CASE eHomeSeq OF
    E_HomingRoutines.eHomeToRef_Bwd:
        stDetectDirection := mcNegativeDirection;
        fbFinishHoming.Distance := fHomeFinishDistance;
    E_HomingRoutines.eHomeToRef_Fwd:
        stDetectDirection := mcPositiveDirection;
        fbFinishHoming.Distance := -fHomeFinishDistance;
END_CASE
bViaLimitSwitch := FALSE;

fbStepAbsoluteSwitchDetection.Options.DisableDriveAccess := stOptions.DisableDriveAccess;
fbStepAbsoluteSwitchDetection(
    Axis := Axis,
    Execute := bDetectionFB_Execute,
    Parameter := stHomingParameter,
    Direction := stDetectDirection,
    SwitchMode := stConfig.stHomingConfig.eRefSwitchMode,
    ReferenceSignal := stRefSwitchSignal,
    Velocity := fVelocityFromCam,
    PositiveLimitSwitch := NOT(bLimitFwd),
    NegativeLimitSwitch := NOT(bLimitBwd),
    Options := stOptions,
    Done => bDetectionFB_Done,
    Busy => bDetectionFB_Busy,
    CommandAborted => bDetectionFB_CommandAborted,
    Error => bDetectionFB_Error,
    ErrorID => nDetectionFB_ErrorID,
    RecordedPosition => fRecordedPosition);
END_ACTION

END_FUNCTION_BLOCK

// ---- tc_mca_std_lib/POUs/Pneumatics/FB_PneumaticAxis.TcPOU

FUNCTION_BLOCK FB_PneumaticAxis

VAR_IN_OUT
    stPneumaticAxisStruct: ST_PneumaticAxisStruct;
END_VAR
VAR
    fbTimerExtend: TON; //Timing the extraction of the cylinder
    fbTimerRetract: TON; //Timing the retraction of the cylinder
    fbTrigRisingEdgePermit: R_TRIG; //Rising edge detection for Permit signal
    fbTrigExtendManual: R_TRIG; //Rising edge detection for manual push button
    fbTrigRetractManual: R_TRIG; //Rising edge detection for manual push button
    bStateChange: BOOL := FALSE; //State of the cylinder changed from extend to retract and vice versa
    bStartExtendManual: BOOL; //Variable to control the solenoid valve with momentary push button
    bStartRetractManual: BOOL; //VAriable to control the solenoid valve with momentary push button
END_VAR


Initialization();

CASE stPneumaticAxisStruct.ePneumaticAxisMode OF

    E_PneumaticMode.eSingleSolenoidControl:
    Single_Solenoid();

    E_PneumaticMode.eError:
    Single_Solenoid_Error();

    E_PneumaticMode.eReset:
    Reset();
END_CASE

ACTION ErrorCheck:
//IF the command to extract is given, but the cylinder hasn't moved from the bEndSwitchBwd
    IF  fbTimerExtend.Q AND stPneumaticAxisStruct.stPneumaticAxisStatus.bRetracted THEN
             stPneumaticAxisStruct.stPneumaticAxisStatus.bExtending := FALSE;
             stPneumaticAxisStruct.ePneumaticAxisMode := E_PneumaticMode.eError;
    END_IF
//If the command to extract has timed out
    IF  fbTimerExtend.Q AND (NOT stPneumaticAxisStruct.stPneumaticAxisStatus.bRetracted AND NOT stPneumaticAxisStruct.stPneumaticAxisStatus.bExtended) THEN
            stPneumaticAxisStruct.stPneumaticAxisStatus.bExtending := FALSE;
            stPneumaticAxisStruct.ePneumaticAxisMode := E_PneumaticMode.eError;
    END_IF

//IF the command to retract has been given, but the cylinder hasn't moved from bEndSwitchFwd
        IF  fbTimerRetract.Q AND stPneumaticAxisStruct.stPneumaticAxisStatus.bExtended THEN
            stPneumaticAxisStruct.stPneumaticAxisStatus.bRetracting := FALSE;
            stPneumaticAxisStruct.ePneumaticAxisMode := E_PneumaticMode.eError;
        END_IF

//If the command to retract has timed out
        IF  fbTimerRetract.Q AND (NOT stPneumaticAxisStruct.stPneumaticAxisStatus.bExtended AND NOT stPneumaticAxisStruct.stPneumaticAxisStatus.bRetracted) THEN
            stPneumaticAxisStruct.stPneumaticAxisStatus.bRetracting := FALSE;
            stPneumaticAxisStruct.ePneumaticAxisMode := E_PneumaticMode.eError;
        END_IF
END_ACTION

ACTION Initialization:
//Set the inputs of limit switches to bExtracted and bRetracted states of the pneumatic cylinders
stPneumaticAxisStruct.stPneumaticAxisStatus.bRetracted := stPneumaticAxisStruct.stPneumaticAxisInputs.bEndSwitchBwd;
stPneumaticAxisStruct.stPneumaticAxisStatus.bExtended := stPneumaticAxisStruct.stPneumaticAxisInputs.bEndSwitchFwd;
stPneumaticAxisStruct.stPneumaticAxisStatus.bSolenoidActive := stPneumaticAxisStruct.stPneumaticAxisInputs.bSolenoidActive;
stPneumaticAxisStruct.stPneumaticAxisStatus.bPSSPermitOK := stPneumaticAxisStruct.stPneumaticAxisInputs.bPSSPermit;
stPneumaticAxisStruct.stPneumaticAxisStatus.bInterlocked := stPneumaticAxisStruct.stPneumaticAxisControl.bInterlock;


//Check if Permit signal is ON
IF NOT stPneumaticAxisStruct.stPneumaticAxisInputs.bPSSPermit THEN
            stPneumaticAxisStruct.stPneumaticAxisOutputs.bValveOn := FALSE;
            stPneumaticAxisStruct.ePneumaticAxisMode := E_PneumaticMode.eError;
END_IF

//Reset Error
fbTrigRisingEdgePermit(clk:=stPneumaticAxisStruct.stPneumaticAxisControl.bReset);

IF fbTrigRisingEdgePermit.Q THEN
    stPneumaticAxisStruct.ePneumaticAxisMode := E_PneumaticMode.eReset;
END_IF

//Check if Interlock signal is ON
IF stPneumaticAxisStruct.stPneumaticAxisControl.bInterlock THEN
            stPneumaticAxisStruct.stPneumaticAxisOutputs.bValveOn := FALSE;
            stPneumaticAxisStruct.ePneumaticAxisMode := E_PneumaticMode.eError;
END_IF

//Check for errors in Air pressure (to be implemented)
END_ACTION

ACTION Reset:
//Reset all the error messages
//Set the operating mode to Single Solenoid Control

stPneumaticAxisStruct.stPneumaticAxisStatus.sStatus := 'NO_ERRORS_READY_TO_START';
stPneumaticAxisStruct.ePneumaticAxisErrors := E_PneumaticAxisErrors.eNoError;
stPneumaticAxisStruct.stPneumaticAxisStatus.bError := FALSE;
stPneumaticAxisStruct.ePneumaticAxisMode := E_PneumaticMode.eSingleSolenoidControl;
END_ACTION

ACTION Single_Solenoid:
//Enter allowed times for extraction and retraction of pneumatic cylinder in seconds
 fbTimerExtend.PT := INT_TO_TIME( stPneumaticAxisStruct.stPneumaticAxisConfig.nTimeToExtend)*1000;
 fbTimerRetract.PT := INT_TO_TIME( stPneumaticAxisStruct.stPneumaticAxisConfig.nTimeToRetract)*1000;


//Starting the timing of extraction movement
fbTimerExtend();
fbTimerExtend(IN := stPneumaticAxisStruct.stPneumaticAxisStatus.bExtending);

//If the manual momentary push button is used for control of the pneumatic cylinder
fbTrigExtendManual(clk:=stPneumaticAxisStruct.stPneumaticAxisInputs.bOpenManual);

IF fbTrigExtendManual.Q THEN
    bStartExtendManual := TRUE;
END_IF

//Starting the extraction movement
IF (stPneumaticAxisStruct.stPneumaticAxisControl.bExtend OR bStartExtendManual) THEN
        stPneumaticAxisStruct.stPneumaticAxisOutputs.bValveOn := TRUE;
        stPneumaticAxisStruct.stPneumaticAxisStatus.bExtending := TRUE;
//If the command to retract is given while the cylinder is extracting
    IF NOT stPneumaticAxisStruct.stPneumaticAxisStatus.bExtended AND NOT stPneumaticAxisStruct.stPneumaticAxisStatus.bRetracted THEN
        IF (stPneumaticAxisStruct.stPneumaticAxisControl.bRetract OR bStartRetractManual) THEN
            stPneumaticAxisStruct.stPneumaticAxisOutputs.bValveOn := FALSE;
            stPneumaticAxisStruct.stPneumaticAxisStatus.bRetracting := TRUE;
            stPneumaticAxisStruct.stPneumaticAxisStatus.bExtending := FALSE;
            stPneumaticAxisStruct.stPneumaticAxisControl.bExtend := FALSE;
        bStartExtendManual := FALSE;
        END_IF
    END_IF


END_IF
//Check for errors while the cylinder is extending
ErrorCheck();

// Extraction of the cylinder finished, reset timer
IF (stPneumaticAxisStruct.stPneumaticAxisControl.bExtend OR bStartExtendManual) AND stPneumaticAxisStruct.stPneumaticAxisStatus.bExtended THEN
        bStateChange := TRUE;
        stPneumaticAxisStruct.stPneumaticAxisStatus.bExtending := FALSE;
        stPneumaticAxisStruct.stPneumaticAxisControl.bExtend := FALSE;
        bStartExtendManual := FALSE;
END_IF



//Starting the retraction movement and retraction timing
fbTimerRetract();
fbTimerRetract (IN := stPneumaticAxisStruct.stPneumaticAxisStatus.bRetracting);

//If the manual momentary push button is used for control of the pneumatic cylinder
fbTrigRetractManual(clk:=stPneumaticAxisStruct.stPneumaticAxisInputs.bCloseManual);

IF fbTrigRetractManual.Q THEN
    bStartRetractManual := TRUE;
END_IF

IF (stPneumaticAxisStruct.stPneumaticAxisControl.bRetract OR bStartRetractManual) THEN
        stPneumaticAxisStruct.stPneumaticAxisOutputs.bValveOn := FALSE;
        stPneumaticAxisStruct.stPneumaticAxisStatus.bRetracting := TRUE;


END_IF
//Check for errors while the cylinder is retracting
ErrorCheck();
// Retraction of the cylinder finished, reset timer
IF  (stPneumaticAxisStruct.stPneumaticAxisControl.bRetract OR bStartRetractManual) AND stPneumaticAxisStruct.stPneumaticAxisStatus.bRetracted THEN
        bStateChange := FALSE;
        stPneumaticAxisStruct.stPneumaticAxisStatus.bRetracting := FALSE;
        stPneumaticAxisStruct.stPneumaticAxisControl.bRetract := FALSE;
        bStartRetractManual := FALSE;
END_IF
END_ACTION

ACTION Single_Solenoid_Error:
IF NOT stPneumaticAxisStruct.stPneumaticAxisInputs.bPSSPermit THEN
    stPneumaticAxisStruct.ePneumaticAxisErrors := E_PneumaticAxisErrors.eNoPSSPermit;
END_IF

IF stPneumaticAxisStruct.stPneumaticAxisControl.bInterlock THEN
     stPneumaticAxisStruct.ePneumaticAxisErrors := E_PneumaticAxisErrors.eInterlockOn;
END_IF

IF  fbTimerExtend.Q AND stPneumaticAxisStruct.stPneumaticAxisStatus.bRetracted THEN
    stPneumaticAxisStruct.ePneumaticAxisErrors := E_PneumaticAxisErrors.eNotMovingExtract;
END_IF

IF  fbTimerExtend.Q AND NOT stPneumaticAxisStruct.stPneumaticAxisStatus.bRetracted AND NOT stPneumaticAxisStruct.stPneumaticAxisStatus.bExtended THEN
    stPneumaticAxisStruct.ePneumaticAxisErrors := E_PneumaticAxisErrors.eExtractTimedOut;
END_IF

IF  fbTimerRetract.Q AND stPneumaticAxisStruct.stPneumaticAxisStatus.bExtended THEN
    stPneumaticAxisStruct.ePneumaticAxisErrors := E_PneumaticAxisErrors.eNotMovingRetract;
END_IF

IF  fbTimerRetract.Q AND NOT stPneumaticAxisStruct.stPneumaticAxisStatus.bExtended AND NOT stPneumaticAxisStruct.stPneumaticAxisStatus.bRetracted THEN
    stPneumaticAxisStruct.ePneumaticAxisErrors := E_PneumaticAxisErrors.eRetractTimedOut;
END_IF


CASE  stPneumaticAxisStruct.ePneumaticAxisErrors OF

    E_PneumaticAxisErrors.eNoError:
    stPneumaticAxisStruct.stPneumaticAxisStatus.bError := FALSE;

    E_PneumaticAxisErrors.eExtractTimedOut:
    stPneumaticAxisStruct.stPneumaticAxisStatus.sStatus := 'ERROR: COMMAND TIMED OUT';
    stPneumaticAxisStruct.stPneumaticAxisStatus.bError := TRUE;

    E_PneumaticAxisErrors.eRetractTimedOut:
    stPneumaticAxisStruct.stPneumaticAxisStatus.sStatus := 'ERROR: COMMAND TIMED OUT';
    stPneumaticAxisStruct.stPneumaticAxisStatus.bError := TRUE;

    E_PneumaticAxisErrors.eNotMovingExtract:
    stPneumaticAxisStruct.stPneumaticAxisStatus.sStatus := 'ERROR: CYLINDER NOT MOVING';
    stPneumaticAxisStruct.stPneumaticAxisStatus.bError := TRUE;

    E_PneumaticAxisErrors.eNotMovingRetract:
    stPneumaticAxisStruct.stPneumaticAxisStatus.sStatus := 'ERROR: CYLINDER NOT MOVING';
    stPneumaticAxisStruct.stPneumaticAxisStatus.bError := TRUE;

    E_PneumaticAxisErrors.eNoPSSPermit:
    stPneumaticAxisStruct.stPneumaticAxisStatus.sStatus := 'ERROR: NO PERMIT SIGNAL';
    stPneumaticAxisStruct.stPneumaticAxisStatus.bError := TRUE;

    E_PneumaticAxisErrors.eInterlockOn:
    stPneumaticAxisStruct.stPneumaticAxisStatus.sStatus := 'ERROR: INTERLOCK SIGNAL ON';
    stPneumaticAxisStruct.stPneumaticAxisStatus.bError := TRUE;

END_CASE

stPneumaticAxisStruct.stPneumaticAxisControl.bExtend := FALSE;
stPneumaticAxisStruct.stPneumaticAxisControl.bRetract := FALSE;
stPneumaticAxisStruct.stPneumaticAxisOutputs.bValveOn := FALSE;
bStartExtendManual := FALSE;
bStartRetractManual := FALSE;
stPneumaticAxisStruct.stPneumaticAxisStatus.bExtending := FALSE;
stPneumaticAxisStruct.stPneumaticAxisStatus.bRetracting := FALSE;
END_ACTION

END_FUNCTION_BLOCK

// ---- POUs/Application_Specific/Axes/Axis_Template.TcPOU
PROGRAM Axis_Template
VAR
//Outputs: Power for Limit switches, Home Sensors, etc.
    //bPowerSwitchesAxis1 AT %Q*: BOOL:= TRUE;

//Hardware interlocks
    //bInterlockFwdOK AT %I*: BOOL;
END_VAR

//Initial parameters of an Axis
(* Uncomment the next IF statement to configure and activate the intial parameters of the axis
IF _TaskInfo[fbGetCurTaskIndex.index].FirstCycle THEN
    //Axis description for EPICS PV
    GVL.astAxes[x].stDescription.sAxisName := 'MotorApplication1';
    GVL.astAxes[x].stDescription.eUnit := E_AxisEngUnit.eMeter;
    GVL.astAxes[x].stDescription.nPrefix := -3;

    //Initial default values:
    GVL.astAxes[x].stConfig.eHomeSeq := 0;
    GVL.astAxes[x].stConfig.fHomePosition := 0.0;
    GVL.astAxes[x].stConfig.fHomeFinishDistance := 0.0;
    GVL.astAxes[x].stConfig.eRestorePosition := E_RestorePosition.eRestoreWithoutHome;

    GVL.astAxes[x].stConfig.bEnableTemperatureDisable := FALSE;
    GVL.astAxes[x].stConfig.fMaxTemperature := 0.0;
END_IF
*)
//Define ACTIONS() or write exclusive code for an specific axis.
(*Eg. Stop when temperature reaches certain values, reduce speed if  a signal is activated, etc.
Eg. GVL.astAxes[x].stControl.bInterlockFwd := NOT bInterlockFwdOK;*)

END_PROGRAM

// ---- POUs/Application_Specific/Applications/Application_Template.TcPOU
PROGRAM Application_Template
VAR
    //Define all necessary variables for your application

END_VAR

//Program any specific code or safety code for an specific application when it involves multiple axes
//Eg. Collision avoidance, interlocks, sequencing, etc.

END_PROGRAM

// ---- POUs/Application_Specific/Axes/Pneumatics_Template.TcPOU
PROGRAM Pneumatics_Template
VAR
END_VAR

//Test the program to control pneumatic acutator through PneumaticsVisu.
//Currently implemented control of single solenoid through PLC and and manually, with two momentary push buttons.

END_PROGRAM

// ---- tc_mca_std_lib/POUs/FB_ESSMonitoring.TcPOU

FUNCTION_BLOCK FB_ESSMonitoring
VAR_INPUT
    nEcMasterNetId: T_AmsNetId;
END_VAR
VAR_OUTPUT
    aErrorID: ARRAY [1..nMaxAlarms] OF INT;
    aErrorMsg: ARRAY [1..nMaxAlarms] OF STRING;
    nEcMasterFramesLost: UDINT;
    nCPULoad: UDINT;
    fCycleExecTime_ms: REAL;
    nAlarmGrpBitNumber: UDINT;
END_VAR
VAR
    //Outputs
    bFan1 AT %Q*: BOOL := TRUE;
    bFan2 AT %Q*: BOOL := TRUE;
    bDCSupplyLED AT %Q*: BOOL := TRUE;
    bAcknowledgeLED AT %Q*: BOOL;
    bStatusLED AT %Q*: BOOL;
    bWarningLED AT %Q*: BOOL;
    bEmergencyLED AT %Q*: BOOL;
    //Inputs
    b24VDC1_OK AT %I*: BOOL;
    b24VDC2_OK AT %I*: BOOL;
    b48VDC1_OK AT %I*: BOOL;
    bFuse1_OK AT %I*: BOOL;
    bFuse2_OK AT %I*: BOOL;
    bFuse3_OK AT %I*: BOOL;
    bFuse4_OK AT %I*: BOOL;
    bFuse5_OK AT %I*: BOOL;
    bFuse6_OK AT %I*: BOOL;
    bFuse7_OK AT %I*: BOOL;
    bFuse8_OK AT %I*: BOOL;
    bSafety_OK AT %I*: BOOL;
    bFan1_OK AT %I*: BOOL;
    bFan2_OK AT %I*: BOOL;
    nTemp1 AT %I*: INT;
    nTemp2 AT %I*: INT;
    nEcMasterDevState AT %I*: UINT;
    aAlarmList: ARRAY [1..nMaxAlarms] OF ST_MonitoringAlarm := [
                    (*[1]*)(nStatusLED:=E_MonitoringLedFunction.eFast, nWarningLED:=E_MonitoringLedFunction.eUndefined, nEmergencyLED:=E_MonitoringLedFunction.eSteady, nAcknowledgeLED:=E_MonitoringLedFunction.eUndefined, nErrorID:=1 ,sErrorMsg:='The DC OK Status from PS or DC-DC converter 24V-1 is OFF.'),
                    (*[2]*)(nStatusLED:=E_MonitoringLedFunction.eUndefined, nWarningLED:=E_MonitoringLedFunction.eUndefined, nEmergencyLED:=E_MonitoringLedFunction.eUndefined, nAcknowledgeLED:=E_MonitoringLedFunction.eUndefined, nErrorID:=2 ,sErrorMsg:='The DC OK Status from PS 24V-2 is OFF.'),
                    (*[3]*)(nStatusLED:=E_MonitoringLedFunction.eFast, nWarningLED:=E_MonitoringLedFunction.eUndefined, nEmergencyLED:=E_MonitoringLedFunction.eSteady, nAcknowledgeLED:=E_MonitoringLedFunction.eUndefined, nErrorID:=4 ,sErrorMsg:='The DC OK Status from PS 48V-1 is OFF.'),
                    (*[4]*)(nStatusLED:=E_MonitoringLedFunction.eUndefined, nWarningLED:=E_MonitoringLedFunction.eUndefined, nEmergencyLED:=E_MonitoringLedFunction.eUndefined, nAcknowledgeLED:=E_MonitoringLedFunction.eUndefined, nErrorID:=8 ,sErrorMsg:='Output 1 on LOCC box 1 tripped'),
                    (*[5]*)(nStatusLED:=E_MonitoringLedFunction.eSlow, nWarningLED:=E_MonitoringLedFunction.eUndefined, nEmergencyLED:=E_MonitoringLedFunction.eSteady, nAcknowledgeLED:=E_MonitoringLedFunction.eUndefined, nErrorID:=9 ,sErrorMsg:='Output 2 on LOCC box 1 tripped'),
                    (*[6]*)(nStatusLED:=E_MonitoringLedFunction.eUndefined, nWarningLED:=E_MonitoringLedFunction.eUndefined, nEmergencyLED:=E_MonitoringLedFunction.eUndefined, nAcknowledgeLED:=E_MonitoringLedFunction.eUndefined, nErrorID:=10 ,sErrorMsg:='Output 1 on LOCC box 2 tripped'),
                    (*[7]*)(nStatusLED:=E_MonitoringLedFunction.eSlow, nWarningLED:=E_MonitoringLedFunction.eUndefined, nEmergencyLED:=E_MonitoringLedFunction.eSteady, nAcknowledgeLED:=E_MonitoringLedFunction.eUndefined, nErrorID:=11 ,sErrorMsg:='Output 2 on LOCC box 2 tripped'),
                    (*[8]*)(nStatusLED:=E_MonitoringLedFunction.eSteady, nWarningLED:=E_MonitoringLedFunction.eSteady, nEmergencyLED:=E_MonitoringLedFunction.eUndefined, nAcknowledgeLED:=E_MonitoringLedFunction.eUndefined, nErrorID:=12 ,sErrorMsg:='Output 1 on LOCC box 3 tripped'),
                    (*[9]*)(nStatusLED:=E_MonitoringLedFunction.eSteady, nWarningLED:=E_MonitoringLedFunction.eSteady, nEmergencyLED:=E_MonitoringLedFunction.eUndefined, nAcknowledgeLED:=E_MonitoringLedFunction.eUndefined, nErrorID:=13 ,sErrorMsg:='Output 2 on LOCC box 3 tripped'),
                    (*[10]*)(nStatusLED:=E_MonitoringLedFunction.eSlow, nWarningLED:=E_MonitoringLedFunction.eSteady, nEmergencyLED:=E_MonitoringLedFunction.eUndefined, nAcknowledgeLED:=E_MonitoringLedFunction.eUndefined, nErrorID:=14 ,sErrorMsg:='LOCC box 4 or single DC breaker 1 tripped'),
                    (*[11]*)(nStatusLED:=E_MonitoringLedFunction.eSlow, nWarningLED:=E_MonitoringLedFunction.eSteady, nEmergencyLED:=E_MonitoringLedFunction.eUndefined, nAcknowledgeLED:=E_MonitoringLedFunction.eUndefined, nErrorID:=15 ,sErrorMsg:='LOCC box 5 or single DC breaker 2 tripped'),
                    (*[12]*)(nStatusLED:=E_MonitoringLedFunction.eUndefined, nWarningLED:=E_MonitoringLedFunction.eSteady, nEmergencyLED:=E_MonitoringLedFunction.eUndefined, nAcknowledgeLED:=E_MonitoringLedFunction.eUndefined, nErrorID:=21 ,sErrorMsg:='Speed of Fan 1 below a critical limit'),
                    (*[13]*)(nStatusLED:=E_MonitoringLedFunction.eUndefined, nWarningLED:=E_MonitoringLedFunction.eSteady, nEmergencyLED:=E_MonitoringLedFunction.eUndefined, nAcknowledgeLED:=E_MonitoringLedFunction.eUndefined, nErrorID:=22 ,sErrorMsg:='Speed of Fan 2 below a critical limit'),
                    (*[14]*)(nStatusLED:=E_MonitoringLedFunction.eUndefined, nWarningLED:=E_MonitoringLedFunction.eSteady, nEmergencyLED:=E_MonitoringLedFunction.eSteady, nAcknowledgeLED:=E_MonitoringLedFunction.eUndefined, nErrorID:=23 ,sErrorMsg:='Temperature 1 too high' ),
                    (*[15]*)(nStatusLED:=E_MonitoringLedFunction.eUndefined, nWarningLED:=E_MonitoringLedFunction.eSteady, nEmergencyLED:=E_MonitoringLedFunction.eSteady, nAcknowledgeLED:=E_MonitoringLedFunction.eUndefined, nErrorID:=24 ,sErrorMsg:='Temperature 2 too high'),
                    (*[16]*)(nStatusLED:=E_MonitoringLedFunction.eSteady, nWarningLED:=E_MonitoringLedFunction.eSteady, nEmergencyLED:=E_MonitoringLedFunction.eUndefined, nAcknowledgeLED:=E_MonitoringLedFunction.eUndefined, nErrorID:=30 ,sErrorMsg:='Safety relay 1 triggered'),
                    (*[17]*)(nStatusLED:=E_MonitoringLedFunction.eSteady, nWarningLED:=E_MonitoringLedFunction.eSlow, nEmergencyLED:=E_MonitoringLedFunction.eUndefined, nAcknowledgeLED:=E_MonitoringLedFunction.eUndefined, nErrorID:=101 ,sErrorMsg:='EtherCAT Master is not ok'),
                    (*[18]*)(nStatusLED:=E_MonitoringLedFunction.eSteady, nWarningLED:=E_MonitoringLedFunction.eSlow, nEmergencyLED:=E_MonitoringLedFunction.eSteady, nAcknowledgeLED:=E_MonitoringLedFunction.eUndefined, nErrorID:=102 ,sErrorMsg:='At least one EtherCAT slave is not in OP state'),
                    (*[19]*)(nStatusLED:=E_MonitoringLedFunction.eSteady, nWarningLED:=E_MonitoringLedFunction.eSlow, nEmergencyLED:=E_MonitoringLedFunction.eSteady, nAcknowledgeLED:=E_MonitoringLedFunction.eUndefined, nErrorID:=103 ,sErrorMsg:='At least one EtherCAT slave link is faulted'),
                    (*[20]*)(nStatusLED:=E_MonitoringLedFunction.eSteady, nWarningLED:=E_MonitoringLedFunction.eSlow, nEmergencyLED:=E_MonitoringLedFunction.eUndefined, nAcknowledgeLED:=E_MonitoringLedFunction.eUndefined, nErrorID:=104 ,sErrorMsg:='Overflow in PLC cycle time'),
                    (*[21]*)(nStatusLED:=E_MonitoringLedFunction.eSteady, nWarningLED:=E_MonitoringLedFunction.eSlow, nEmergencyLED:=E_MonitoringLedFunction.eUndefined, nAcknowledgeLED:=E_MonitoringLedFunction.eUndefined, nErrorID:=105 ,sErrorMsg:='CPU Load High')];

    aTempErrorID: ARRAY [1..nMaxAlarms] OF INT;
    aTempErrorMsg: ARRAY [1..nMaxAlarms] OF STRING;
    nLEDAlarmID: INT;
    sLEDAlarmMsg: STRING;
    nAlarmCnt: INT;
    nAlarmBitNumber: UDINT;

    bCPUOverloaded: BOOL;
    bEcMasterNotOK: BOOL;
    bSlaveStateNotOP: BOOL;
    bSlaveLinkNotOK: BOOL;
    bCycleTimeExceeded: BOOL;
    //Cpu Monitor
    fbMonitorCPU: TC_CpuUsage;
    fbUpdateCPULoadTON: TON;
    fMaxCPULoad: USINT := 85;
    //Ehtercat master device state
    bEcLinkError: BOOL;
    bEcIOlocked: BOOL;
    bEcLinkErrorRedundancyAdapter: BOOL;
    bEcMissingFrame: BOOL;
    bEcOutofSendResources: BOOL;
    bEcWatchdogTriggered: BOOL;
    bEcEthernetDriverNotFound: BOOL;
    bEcIOresetActive: BOOL;
    bEcSlaveINIT: BOOL;
    bEcSlavePreOP: BOOL;
    bEcSlaveSafeOP: BOOL;
    bEcSlaveError: BOOL;
    bEcDCnotInSync: BOOL;
    //Ehtercat slave device state
    fbUpdateEcSlaveStateTON: TON;
    fbGetEcSlaveStates: FB_EcGetAllSlaveStates;
    stSlaveState: ARRAY[0..nMaxECSlaves] OF ST_EcSlaveState;
    nActualEcSlaves: INT := 0;
    i: INT;
    //Frame statistics
    fbUpdateEcMasterFrame: TON;
    fbGetEcMasterFrames: FB_EcMasterFrameStatistic;

    nAcknowledgeLED: E_MonitoringLedFunction;
    nStatusLED: E_MonitoringLedFunction;
    nWarningLED: E_MonitoringLedFunction;
    nEmergencyLED: E_MonitoringLedFunction;
    fbFastBlinkOn: TON;
    fbFastBlinkOff: TON;
    bFastBlink: BOOL;
    fbSlowBlinkOn: TON;
    fbSlowBlinkOff: TON;
    bSlowBlink: BOOL;
END_VAR
VAR CONSTANT
    nMaxAlarms: INT := 50;
    nMaxECSlaves: INT := 255;
    nMaxTemp: INT := 10000;
END_VAR


actMonitorAlarms();
actMonitorCPU();
actMonitorEtherCAT();

ACTION actMonitorAlarms:

aAlarmList[1].bAlarmSet := NOT b24VDC1_OK;
aAlarmList[1].bAlarmReset:= TRUE;
aAlarmList[2].bAlarmSet := b24VDC2_OK;
aAlarmList[2].bAlarmReset:= TRUE;
aAlarmList[3].bAlarmSet := NOT b48VDC1_OK;
aAlarmList[3].bAlarmReset:= TRUE;
aAlarmList[4].bAlarmSet := bFuse1_OK;
aAlarmList[4].bAlarmReset:= TRUE;
aAlarmList[5].bAlarmSet :=  bFuse2_OK;
aAlarmList[5].bAlarmReset:= TRUE;
aAlarmList[6].bAlarmSet := bFuse3_OK;
aAlarmList[6].bAlarmReset:= TRUE;
aAlarmList[7].bAlarmSet := bFuse4_OK;
aAlarmList[7].bAlarmReset:= TRUE;
aAlarmList[8].bAlarmSet := bFuse5_OK;
aAlarmList[8].bAlarmReset:= TRUE;
aAlarmList[9].bAlarmSet := bFuse6_OK;
aAlarmList[9].bAlarmReset:= TRUE;
aAlarmList[10].bAlarmSet := bFuse7_OK;
aAlarmList[10].bAlarmReset:= TRUE;
aAlarmList[11].bAlarmSet := bFuse8_OK;
aAlarmList[11].bAlarmReset:= TRUE;
aAlarmList[12].bAlarmSet := NOT bFan1_OK;
aAlarmList[12].bAlarmReset:= TRUE;
aAlarmList[13].bAlarmSet := NOT bFan2_OK;
aAlarmList[13].bAlarmReset:= TRUE;
aAlarmList[14].bAlarmSet := nTemp1 > nMaxTemp;
aAlarmList[14].bAlarmReset:= TRUE;
aAlarmList[15].bAlarmSet := nTemp2 > nMaxTemp;
aAlarmList[15].bAlarmReset:= TRUE;
aAlarmList[16].bAlarmSet := NOT bSafety_OK;
aAlarmList[16].bAlarmReset:= TRUE;
aAlarmList[17].bAlarmSet := bEcMasterNotOK;
aAlarmList[17].bAlarmReset:= TRUE;
aAlarmList[18].bAlarmSet := bSlaveStateNotOP;
aAlarmList[18].bAlarmReset:= TRUE;
aAlarmList[19].bAlarmSet := bSlaveLinkNotOK;
aAlarmList[19].bAlarmReset:= TRUE;
aAlarmList[20].bAlarmSet := bCycleTimeExceeded;
aAlarmList[20].bAlarmReset:= TRUE;
aAlarmList[21].bAlarmSet := bCPUOverloaded;
aAlarmList[21].bAlarmReset:= TRUE;

FOR i:=1 TO nMaxAlarms DO
    mAlarm(stAlarmData:= aAlarmList[i]);
    IF i = 1 THEN
        nAlarmCnt := 0;
        nAlarmBitNumber := 0;
        MEMSET(ADR(aTempErrorID), 0, SIZEOF(aTempErrorID));
        MEMSET(ADR(aTempErrorMsg), 0, SIZEOF(aTempErrorMsg));
    ELSIF i = nMaxAlarms THEN
        aErrorID := aTempErrorID;
        aErrorMsg := aTempErrorMsg;
        nAlarmGrpBitNumber := nAlarmBitNumber;
    END_IF

    IF aAlarmList[i].bAlarmActive THEN
        nAlarmCnt := nAlarmCnt + 1;
        aTempErrorID[nAlarmCnt] := aAlarmList[i].nErrorID;
        aTempErrorMsg[nAlarmCnt] := aAlarmList[i].sErrorMsg;
        IF nLEDAlarmID = 0 OR (nWarningLED = E_MonitoringLedFunction.eUndefined AND nEmergencyLED = E_MonitoringLedFunction.eUndefined AND aAlarmList[i].nWarningLED > E_MonitoringLedFunction.eUndefined) OR (nEmergencyLED = E_MonitoringLedFunction.eUndefined AND aAlarmList[i].nEmergencyLED > E_MonitoringLedFunction.eUndefined) THEN
            nLEDAlarmID := i;
            sLEDAlarmMsg := aAlarmList[i].sErrorMsg;
            nEmergencyLED := aAlarmList[i].nEmergencyLED;
            nWarningLED := aAlarmList[i].nWarningLED;
            nStatusLED := aAlarmList[i].nStatusLED;
            nAcknowledgeLED := aAlarmList[i].nAcknowledgeLED;
        END_IF
        CASE aAlarmList[i].nErrorID OF
            1,4:
            nAlarmBitNumber.0 := TRUE;
            9,12,13:
            nAlarmBitNumber.1 := TRUE;
            10,11:
            nAlarmBitNumber.2 := TRUE;
            14,15:
            nAlarmBitNumber.3 := TRUE;
            21,22:
            nAlarmBitNumber.4 := TRUE;
            23,24:
            nAlarmBitNumber.5 := TRUE;
            104,105:
            nAlarmBitNumber.6 := TRUE;
            103:
            nAlarmBitNumber.7 := TRUE;
            102:
            nAlarmBitNumber.8 := TRUE;
            30:
            nAlarmBitNumber.9 := TRUE;
        END_CASE
    ELSIF NOT aAlarmList[i].bAlarmActive THEN
        IF nLEDAlarmID = i THEN
            nLEDAlarmID := 0;
            sLEDAlarmMsg := '';
            nEmergencyLED := 0;
            nWarningLED := 0;
            nStatusLED := 0;
            nAcknowledgeLED := 0;
        END_IF
    END_IF
END_FOR

fbFastBlinkOn(IN:=NOT fbFastBlinkOff.q , PT:=T#250MS , Q=> , ET=> );
fbFastBlinkOff(IN:=fbFastBlinkOn.Q , PT:=T#250MS , Q=> , ET=> );
bFastBlink := fbFastBlinkOn.q;

fbSlowBlinkOn(IN:=NOT fbSlowBlinkOff.q , PT:=T#750MS , Q=> , ET=> );
fbSlowBlinkOff(IN:=fbSlowBlinkOn.Q , PT:=T#750MS , Q=> , ET=> );
bSlowBlink := fbSlowBlinkOn.q;

bEmergencyLED := (nEmergencyLED = E_MonitoringLedFunction.eSteady) OR (nEmergencyLED = E_MonitoringLedFunction.eFast AND bFastBlink) OR (nEmergencyLED = E_MonitoringLedFunction.eSlow AND bSlowBlink);
bWarningLED := (nWarningLED = E_MonitoringLedFunction.eSteady) OR (nWarningLED = E_MonitoringLedFunction.eFast AND bFastBlink) OR (nWarningLED = E_MonitoringLedFunction.eSlow AND bSlowBlink);
bStatusLED := (nStatusLED = E_MonitoringLedFunction.eSteady) OR (nStatusLED = E_MonitoringLedFunction.eFast AND bFastBlink) OR (nStatusLED = E_MonitoringLedFunction.eSlow AND bSlowBlink);
bAcknowledgeLED := (nAcknowledgeLED = E_MonitoringLedFunction.eSteady) OR (nAcknowledgeLED = E_MonitoringLedFunction.eFast AND bFastBlink) OR (nAcknowledgeLED = E_MonitoringLedFunction.eSlow AND bSlowBlink);
END_ACTION

ACTION actMonitorCPU:

//Cpu Monitor
fbUpdateCPULoadTON(IN:=NOT fbUpdateCPULoadTON.q , PT:=T#100MS , Q=> , ET=> );
fbMonitorCPU(START:=fbUpdateCPULoadTON.q, TMOUT:= T#5S);

bCPUOverloaded := fbMonitorCPU.USAGE > fMaxCPULoad;
nCPULoad := fbMonitorCPU.USAGE;

fCycleExecTime_ms := UDINT_TO_REAL(_TaskInfo[fbGetCurTaskIndex.index].LastExecTime) / 10000;
bCycleTimeExceeded := _TaskInfo[fbGetCurTaskIndex.index].CycleTimeExceeded;
END_ACTION

ACTION actMonitorEtherCAT:

//Read frames
fbUpdateEcMasterFrame(IN:=NOT fbUpdateEcMasterFrame.q , PT:=T#1000MS , Q=> , ET=> );
fbGetEcMasterFrames(sNetId:= nEcMasterNetId, bExecute:= fbUpdateEcMasterFrame.q);

nEcMasterFramesLost := fbGetEcMasterFrames.nLostFrames;


//Check ethercat slave device state
fbUpdateEcSlaveStateTON(IN:=NOT fbUpdateEcSlaveStateTON.q , PT:=T#100MS , Q=> , ET=> );
fbGetEcSlaveStates(sNetId:= nEcMasterNetId, pStateBuf := ADR(stSlaveState), cbBufLen:=SIZEOF(stSlaveState), bExecute:=fbUpdateEcSlaveStateTON.q);
nActualEcSlaves:=UINT_TO_INT(fbGetEcSlaveStates.nSlaves);

FOR i:=0 TO nActualEcSlaves-1 DO
    IF i = 0 THEN
        bSlaveStateNotOP := FALSE;
        bSlaveLinkNotOK := FALSE;
    END_IF
    IF stSlaveState[i].deviceState <> EC_DEVICE_STATE_OP THEN
        bSlaveStateNotOP := TRUE;
    END_IF
    IF stSlaveState[i].linkState <> EC_LINK_STATE_OK THEN
        bSlaveLinkNotOK := TRUE;
    END_IF
END_FOR

//Check ethercat master device state
bEcLinkError := nEcMasterDevState.0;
bEcIOlocked := nEcMasterDevState.1;
bEcLinkErrorRedundancyAdapter := nEcMasterDevState.2;
bEcMissingFrame := nEcMasterDevState.3;
bEcOutofSendResources := nEcMasterDevState.4;
bEcWatchdogTriggered := nEcMasterDevState.5;
bEcEthernetDriverNotFound := nEcMasterDevState.6;
bEcIOresetActive := nEcMasterDevState.7;
bEcSlaveINIT := nEcMasterDevState.8;
bEcSlavePreOP := nEcMasterDevState.9;
bEcSlaveSafeOP := nEcMasterDevState.10;
bEcSlaveError := nEcMasterDevState.11;
bEcDCnotInSync := nEcMasterDevState.12;

bEcMasterNotOK := nEcMasterDevState > 0;
END_ACTION


METHOD mAlarm : BOOL
VAR_IN_OUT
    stAlarmData: ST_MonitoringAlarm;
END_VAR

IF stAlarmData.bAlarmSet THEN
    stAlarmData.bAlarmActive := TRUE;
ELSIF stAlarmData.bAlarmReset THEN
    stAlarmData.bAlarmActive := FALSE;
END_IF
END_METHOD

END_FUNCTION_BLOCK

// ---- tc_mca_std_lib/POUs/Motion/FB_SlitPair.TcPOU

FUNCTION_BLOCK FB_SlitPair
VAR_INPUT
    iBladeNegative: UINT; //Axis ID for negatively positioned blade
    iBladePositive: UINT; //Axis ID for positively positioned blade
    iGapSize: UINT; //Axis ID for the size of gap between slit blades
    iGapCentre: UINT; //Axis ID for the centre position of the gap formed by slit blades
    bEnable: BOOL; //Enable/disable the slit set
    bReset: BOOL; //Reset the slit set
    fEncoderScaling: LREAL := 10000; //default scaling denominator of 10000
    bAutoHome: BOOL := FALSE;
END_VAR
VAR_OUTPUT
    bEnabled: BOOL := FALSE; //Enabled status of function
    bError: BOOL; //Error status of function
    bHoming: BOOL := FALSE; //TRUE if function is homing axes
END_VAR
VAR
    eSlitPairState: E_SlitPairStates := E_SlitPairStates.INIT; //statemachine index

//Internal statuses for logic
    bResetting: BOOL := FALSE; //TRUE if axis going through a reset
    bAxesEnabled: BOOL := FALSE; //TRUE if all axes enabled
    bBladesHomed: BOOL:= FALSE; //TRUE if blade axes are calibrated
    bGapHomed: BOOL:= FALSE; //TRUE if virtual axes are calibrated
    bBladesCoupled: BOOL:= FALSE; //TRUE if both blade axes are coupled
    bBladesUncoupled: BOOL := FALSE; //TRUE if both blade axes are uncoupled
    bAxisErrorsPresent: BOOL := FALSE; //TRUE if error present on any real or virtual axis
    bFunctionInErrorState: BOOL := FALSE; //TRUE if function block is in one of the error related states
    fGapSizePosition: LREAL;
    iGapSizePosition AT %Q*: UDINT := 0;
    fGapCentrePosition: LREAL;
    iGapCentrePosition AT %Q*: UDINT := 0;
    resetCounterTimeout: UINT :=0;
    mcHomeGapSize: MC_Home;
    mcHomeGapCentre: MC_Home;
END_VAR


(* NOTES
For the virtual axis setup, the encoders need their type changed from "simulation encoder" to "Encoder (Universal)".
In addition the scale factor needs to be changed to a numerator of 1 and denominator of fEncoderScaling which is 10,000 by default)
Care needs to be taken with scaling and setup of both real and virtual axes to ensure velocities are not too fast and axes have time to settle before they submit a "complete move"
*)

//Configure homing routine of virtual axes
GVL.astAxes[iGapSize].stConfig.eHomeSeq := E_HomingRoutines.eHomeDirect;
GVL.astAxes[iGapCentre].stConfig.eHomeSeq := E_HomingRoutines.eHomeDirect;

//Run actions for slit set
actErrorHandling(); //Error handling subroutine
actGapLimits(); //Set virtual axis limits to TRUE
actVirtualAxisPositions(); //Virtual axis encoder position subroutine
actRunMethods(); //Update statuses

//Mc_Home FBs configured to clear homing signal
mcHomeGapSize(Axis := astAxes[iGapSize].Axis, HomingMode:=MC_HomingMode.MC_ResetCalibration);
mcHomeGapCentre(Axis:=astAxes[iGapCentre].Axis, HomingMode:=MC_HomingMode.MC_ResetCalibration);
mcHomeGapSize.Execute := FALSE;
mcHomeGapCentre.Execute := FALSE;

CASE eSlitPairState OF
    E_SlitPairStates.INIT:
        IF bAxesEnabled AND bEnable THEN
            eSlitPairState := E_SlitPairStates.INIT_CLEAR_GEARING;
        END_IF

    E_SlitPairStates.INIT_CLEAR_GEARING:
        actClearSlitGearing();
        eSlitPairState := E_SlitPairStates.INIT_GEAROUT_CHECK;

    E_SlitPairStates.INIT_GEAROUT_CHECK: //Check gearOut completion
        IF bBladesUncoupled THEN
            eSlitPairState := E_SlitPairStates.CHECK_HOME_STATUS;
        END_IF

    E_SlitPairStates.CHECK_HOME_STATUS: //If blades are already homed, skip to virtual homing, if blades not homed and autohome enabled then home blades, otherwise wait for blades to be homed
        IF bBladesHomed THEN
            eSlitPairState := E_SlitPairStates.HOME_GAP; //Skip to functioning
        ELSIF bAutoHome THEN
            eSlitPairState := E_SlitPairStates.HOME_BLADES; //If autohome enabled, home the blades
        END_IF

    E_SlitPairStates.HOME_BLADES: //Initiate homing of blade axes. Homing routine must be pre-configured by user
        GVL.astAxes[iBladeNegative].stControl.eCommand := E_MotionFunctions.eHome;
        GVL.astAxes[iBladePositive].stControl.eCommand := E_MotionFunctions.eHome;
        GVL.astAxes[iBladeNegative].stControl.bExecute := TRUE;
        GVL.astAxes[iBladePositive].stControl.bExecute := TRUE;
        bHoming := TRUE;
        eSlitPairState := E_SlitPairStates.CHECK_BLADE_HOME_COMPLETE;

    E_SlitPairStates.CHECK_BLADE_HOME_COMPLETE: //Wait for completion of blade homing routines
        IF bBladesHomed THEN
            eSlitPairState := E_SlitPairStates.HOME_GAP;
            bHoming := FALSE;
        END_IF

    E_SlitPairStates.HOME_GAP: //"Home" the virtual axes
        GVL.astAxes[iGapSize].stConfig.eHomeSeq := E_HomingRoutines.eHomeDirect;
        GVL.astAxes[iGapCentre].stConfig.eHomeSeq := E_HomingRoutines.eHomeDirect;
        GVL.astAxes[iGapSize].stConfig.fHomePosition := fGapSizePosition;
        GVL.astAxes[iGapCentre].stConfig.fHomePosition := fGapCentrePosition;
        GVL.astAxes[iGapSize].stControl.eCommand := E_MotionFunctions.eHome;
        GVL.astAxes[iGapCentre].stControl.eCommand := E_MotionFunctions.eHome;
        GVL.astAxes[iGapSize].stControl.bExecute := TRUE;
        GVL.astAxes[iGapCentre].stControl.bExecute := TRUE;
        eSlitPairState := E_SlitPairStates.CHECK_GAP_HOME_COMPLETE;

    E_SlitPairStates.CHECK_GAP_HOME_COMPLETE: //Wait for virtual homing completion
        IF bGapHomed THEN
            eSlitPairState := E_SlitPairStates.GEARIN_SLITS;
        END_IF

    E_SlitPairStates.GEARIN_SLITS: //Setup gearing
        actSetupSlitGearing();
        eSlitPairState := E_SlitPairStates.CHECK_GEARIN_SLITS_COMPLETE;

    E_SlitPairStates.CHECK_GEARIN_SLITS_COMPLETE: //Wait for gearing complete
        IF bBladesCoupled THEN
            eSlitPairState := E_SlitPairStates.SLITS_OPERATIONAL;
        END_IF

    E_SlitPairStates.SLITS_OPERATIONAL: //SLITS OPERATIONAL - Monitor for any gear outs and re-gear when no busy blades
        bEnabled := TRUE;
        IF NOT bBladesCoupled AND NOT GVL.astAxes[iBladeNegative].stStatus.bBusy AND NOT GVL.astAxes[iBladePositive].stStatus.bBusy THEN
            eSlitPairState := E_SlitPairStates.GEAROUT_BLADES;
        END_IF

    E_SlitPairStates.GEAROUT_BLADES: //Clear amy residual gearing
        actClearSlitGearing();
        eSlitPairState := E_SlitPairStates.CHECK_GEAROUT_COMPLETE;

    E_SlitPairStates.CHECK_GEAROUT_COMPLETE: //Check gearing cleared
        IF bBladesUncoupled THEN
            eSlitPairState := E_SlitPairStates.CLEAR_GAP_CALIBRATION; //Back to homing, this ensures the setpoint position of the axis is updated.
        END_IF

    E_SlitPairStates.CLEAR_GAP_CALIBRATION:
        mcHomeGapSize.Execute := TRUE;
        mcHomeGapCentre.Execute := TRUE;
        IF mcHomeGapSize.Done AND mcHomeGapCentre.Done THEN
            eSlitPairState := E_SlitPairStates.HOME_GAP; //Back to homing, this ensures the setpoint position of the axis is updated.
        END_IF

    E_SlitPairStates.ERROR: //ERROR STATE
        resetCounterTimeout := 0;
        bError := TRUE;
        bEnabled := FALSE;
        IF bReset THEN
            bResetting := TRUE;
            eSlitPairState := E_SlitPairStates.ERROR_GEAROUT;
        END_IF

    E_SlitPairStates.ERROR_GEAROUT: //Try to clear issues
        actClearSlitGearing();
        eSlitPairState := E_SlitPairStates.ERROR_GEAROUT_CHECK;

    E_SlitPairStates.ERROR_GEAROUT_CHECK:
        IF bBladesUncoupled THEN
            eSlitPairState := E_SlitPairStates.ERROR_RESET_AXES; //Back to homing, this ensures the setpoint position of the axis is updated.
        END_IF

    E_SlitPairStates.ERROR_RESET_AXES: //RESET ALL AXES
        GVL.astAxes[iBladeNegative].stControl.bReset := TRUE;
        GVL.astAxes[iBladePositive].stControl.bReset := TRUE;
        GVL.astAxes[iGapSize].stControl.bReset := TRUE;
        GVL.astAxes[iGapCentre].stControl.bReset := TRUE;
        resetCounterTimeout := resetCounterTimeout + 1;
        eSlitPairState := E_SlitPairStates.ERROR_RESET_CHECK;

    E_SlitPairStates.ERROR_RESET_CHECK:
        IF resetCounterTimeout > 10 THEN
            eSlitPairState := E_SlitPairStates.ERROR;
            bResetting := FALSE;
            RETURN;
        END_IF
        IF bAxisErrorsPresent THEN
            eSlitPairState := E_SlitPairStates.ERROR_RESET_AXES;
        ELSE
            eSlitPairState := E_SlitPairStates.INIT;
            bError := FALSE;
            bResetting := FALSE;
        END_IF
END_CASE
bReset := FALSE;

ACTION actClearSlitGearing:
//Action to send gearOut command to blade axes
GVL.astAxes[iBladeNegative].stControl.eCommand := E_MotionFunctions.eGearOut;
GVL.astAxes[iBladePositive].stControl.eCommand := E_MotionFunctions.eGearOut;
GVL.astAxes[iBladeNegative].stControl.bExecute := TRUE;
GVL.astAxes[iBladePositive].stControl.bExecute := TRUE;
END_ACTION

ACTION actErrorHandling:
//Error handling for slit functionality
IF bResetting THEN //ignore setting in error state if FB going through a reset
    RETURN;
END_IF

IF NOT bError AND bAxisErrorsPresent THEN
    eSlitPairState := E_SlitPairStates.ERROR;
END_IF
IF eSlitPairState <> E_SlitPairStates.INIT AND NOT bAxesEnabled THEN
    eSlitPairState := E_SlitPairStates.ERROR;
END_IF
IF (eSlitPairState <> E_SlitPairStates.INIT AND NOT bFunctionInErrorState) AND NOT bEnable THEN
    eSlitPairState := E_SlitPairStates.ERROR;
END_IF
IF bEnabled AND NOT bBladesHomed THEN
    eSlitPairState := E_SlitPairStates.ERROR;
END_IF
END_ACTION

ACTION actGapLimits:
//Set Virtual axis inputs to TRUE to enable movement
GVL.astAxes[iGapSize].stInputs.bLimitBwd := TRUE;
GVL.astAxes[iGapSize].stInputs.bLimitFwd := TRUE;
GVL.astAxes[iGapCentre].stInputs.bLimitBwd := TRUE;
GVL.astAxes[iGapCentre].stInputs.bLimitFwd := TRUE;
END_ACTION

ACTION actRunMethods:
checkAllAxesEnabled(bOutput => bAxesEnabled);
checkBladesHomed(bOutput => bBladesHomed);
checkVirtualHomed(bOutput => bGapHomed);
checkBladesCoupled(bOutput => bBladesCoupled);
checkBladesUncoupled(bOutput => bBladesUncoupled);
checkAllAxisErrors(bOutput => bAxisErrorsPresent);
checkErrorState(bOutput => bFunctionInErrorState);
END_ACTION

ACTION actSetupSlitGearing:
GVL.astAxes[iBladeNegative].stControl.eCommand := E_MotionFunctions.eGearInMultiMaster;
GVL.astAxes[iBladeNegative].stConfig.astMultiMasterAxis[1].nIndex := iGapSize;
GVL.astAxes[iBladeNegative].stConfig.astMultiMasterAxis[1].fRatio := -0.5;
GVL.astAxes[iBladeNegative].stConfig.astMultiMasterAxis[2].nIndex := iGapCentre;
GVL.astAxes[iBladeNegative].stConfig.astMultiMasterAxis[2].fRatio := 1;
GVL.astAxes[iBladePositive].stControl.eCommand := E_MotionFunctions.eGearInMultiMaster;
GVL.astAxes[iBladePositive].stConfig.astMultiMasterAxis[1].nIndex := iGapSize;
GVL.astAxes[iBladePositive].stConfig.astMultiMasterAxis[1].fRatio := 0.5;
GVL.astAxes[iBladePositive].stConfig.astMultiMasterAxis[2].nIndex := iGapCentre;
GVL.astAxes[iBladePositive].stConfig.astMultiMasterAxis[2].fRatio := 1;
GVL.astAxes[iBladeNegative].stControl.bExecute := TRUE;
GVL.astAxes[iBladePositive].stControl.bExecute := TRUE;
END_ACTION

ACTION actVirtualAxisPositions:
(*Calculate virtual axis positions and convert to UDINT.
Conversion to UDINT is prohibited if it would exceed UDINT max value of 4,294,967,295.
If this is not done, it can cause overflow when connected to the encoder input and hard-crash the PLC which will only recover with a power cycle.
To preserve decimal position data of the LREAL (i.e. anything <1mm) it is necessary to scale the value before converting to UDINT.
This can be reversed with the correct scaling at the NC encoder level.
*)
fGapSizePosition := GVL.astAxes[iBladePositive].stStatus.fActPosition - GVL.astAxes[iBladeNegative].stStatus.fActPosition;
fGapCentrePosition := (GVL.astAxes[iBladePositive].stStatus.fActPosition + GVL.astAxes[iBladeNegative].stStatus.fActPosition) / 2;

IF bBladesHomed THEN
    IF ABS(fGapSizePosition) < 100000 THEN
        iGapSizePosition := LREAL_TO_UDINT(fGapSizePosition*fEncoderScaling);
    END_IF
    IF ABS(fGapCentrePosition) < 100000 THEN
        iGapCentrePosition := LREAL_TO_UDINT(fGapCentrePosition*fEncoderScaling);
    END_IF
END_IF
END_ACTION

(*Method to check if all axes (real and virtual) are enabled.
Only returns TRUE if BOTH blades are homed*)
METHOD checkAllAxesEnabled: BOOL
VAR_OUTPUT
    bOutput: BOOL:= TRUE;
END_VAR
IF NOT GVL.astAxes[iBladeNegative].stStatus.bEnabled THEN
    bOutput := FALSE;
END_IF
IF NOT GVL.astAxes[iBladePositive].stStatus.bEnabled THEN
    bOutput := FALSE;
END_IF
IF NOT GVL.astAxes[iGapSize].stStatus.bEnabled THEN
    bOutput := FALSE;
END_IF
IF NOT GVL.astAxes[iGapCentre].stStatus.bEnabled THEN
    bOutput := FALSE;
END_IF
END_METHOD

(*Method to check if an error is present on any axis.
Returns TRUE if an error is present on any axis *)
METHOD checkAllAxisErrors: BOOL
VAR_OUTPUT
    bOutput: BOOL := FALSE;
END_VAR
IF GVL.astAxes[iGapSize].stStatus.bError THEN
    bOutput := TRUE;
END_IF
IF GVL.astAxes[iGapCentre].stStatus.bError THEN
    bOutput := TRUE;
END_IF
IF GVL.astAxes[iBladeNegative].stStatus.bError THEN
    bOutput := TRUE;
END_IF
IF GVL.astAxes[iBladePositive].stStatus.bError THEN
    bOutput := TRUE;
END_IF
END_METHOD

(*Method to check if both blades are coupled to the virtual axes.
Only returns TRUE if BOTH blades are coupled *)
METHOD checkBladesCoupled: BOOL
VAR_OUTPUT
    bOutput: BOOL := TRUE;
END_VAR
IF NOT GVL.astAxes[iBladeNegative].stStatus.bGeared THEN
    bOutput := FALSE;
END_IF
IF NOT GVL.astAxes[iBladePositive].stStatus.bGeared THEN
    bOutput := FALSE;
END_IF
END_METHOD

(*Method to check if blade axes are homed/have the calibration flag.
Only returns TRUE if BOTH blades are homed*)
METHOD checkBladesHomed: BOOL
VAR_OUTPUT
    bOutput: BOOL := TRUE;
END_VAR
IF NOT GVL.astAxes[iBladeNegative].stStatus.bHomed THEN
    bOutput := FALSE;
END_IF
IF NOT GVL.astAxes[iBladePositive].stStatus.bHomed THEN
    bOutput := FALSE;
END_IF
END_METHOD

(*Method to check if both blades are uncoupled from the virtual axes.
Only returns TRUE if BOTH blades are uncoupled *)
METHOD checkBladesUncoupled: BOOL
VAR_OUTPUT
    bOutput: BOOL:= TRUE;
END_VAR
IF GVL.astAxes[iBladeNegative].stStatus.bGeared THEN
    bOutput := FALSE;
END_IF
IF GVL.astAxes[iBladePositive].stStatus.bGeared THEN
    bOutput := FALSE;
END_IF
END_METHOD

METHOD checkErrorState: BOOL
VAR_OUTPUT
    bOutput: BOOL := FALSE;
END_VAR
IF eSlitPairState = E_SlitPairStates.ERROR THEN
    bOutput := TRUE;
END_IF
IF eSlitPairState = E_SlitPairStates.ERROR_GEAROUT THEN
    bOutput := TRUE;
END_IF
IF eSlitPairState = E_SlitPairStates.ERROR_GEAROUT_CHECK THEN
    bOutput := TRUE;
END_IF
IF eSlitPairState = E_SlitPairStates.ERROR_RESET_AXES THEN
    bOutput := TRUE;
END_IF
IF eSlitPairState = E_SlitPairStates.ERROR_RESET_CHECK THEN
    bOutput := TRUE;
END_IF
END_METHOD

(*Method to check if the virtual axes for gap size and gap centre are homed/the calibration flag is present.
Only returns TRUE if BOTH virtual axes are homed *)
METHOD checkVirtualHomed: BOOL
VAR_OUTPUT
    bOutput: BOOL:= TRUE;
END_VAR
IF NOT GVL.astAxes[iGapSize].stStatus.bHomed THEN
    bOutput := FALSE;
END_IF
IF NOT GVL.astAxes[iGapCentre].stStatus.bHomed THEN
    bOutput := FALSE;
END_IF
END_METHOD

END_FUNCTION_BLOCK

// ---- tc_mca_std_lib/POUs/Motion/FB_SlitPairV2.TcPOU

FUNCTION_BLOCK FB_SlitPairV2
VAR_INPUT
    nIdPositiveAxis: UINT; //ID of axis for which positive motion increases gap size
    nIdNegativeAxis: UINT; //ID of axis for which negative motion increases gap size
    nIdGapSizeAxis: UINT; //ID of virtual gap aperture size axis
    nIdGapCentreAxis: UINT; //ID of virtual gap centre position axis

    bEnable: BOOL; //Enable slit pair logic functionality
    bReset: BOOL; //Reset from error state
    fEncoderScaling: LREAL := 10000; //Virtual axis scaling denominator, default of 10000
END_VAR
VAR
    nGapSizeEncoder AT %Q*: UDINT := 0;
    nGapCentreEncoder AT %Q*: UDINT := 0;
    fGapSize: LREAL;
    fGapCentre: LREAL;
    bAllHalted: BOOL := FALSE;
    bInternalResetHome: BOOL :=FALSE;

    fbSetpointGenEnablePositiveAxis: MC_ExtSetPointGenEnable;
    fbSetpointGenEnableNegativeAxis: MC_ExtSetPointGenEnable;
    fbSetpointGenEnableGapSizeAxis: MC_ExtSetPointGenEnable;
    fbSetpointGenEnableGapCentreAxis: MC_ExtSetPointGenEnable;

    fbSetpointGenDisablePositiveAxis: MC_ExtSetPointGenDisable;
    fbSetpointGenDisableNegativeAxis: MC_ExtSetPointGenDisable;
    fbSetpointGenDisableGapSizeAxis: MC_ExtSetPointGenDisable;
    fbSetpointGenDisableGapCentreAxis: MC_ExtSetPointGenDisable;

    fPosSetpointPositiveAxis: LREAL;
    fPosSetpointNegativeAxis: LREAL;
    fPosSetpointGapSizeAxis: LREAL;
    fPosSetpointGapCentreAxis: LREAL;

    fVeloSetpointPositiveAxis: LREAL;
    fVeloSetpointNegativeAxis: LREAL;
    fVeloSetpointGapSizeAxis: LREAL;
    fVeloSetpointGapCentreAxis: LREAL;

    nDirectionPositiveAxis: DINT;
    nDirectionNegativeAxis: DINT;
    nDirectionGapSizeAxis: DINT;
    nDirectionGapCentreAxis: DINT;

    eState: E_SlitPairStatesV2 := E_SlitPairStatesV2.eInit;

    bInternalReset: BOOL;
    bHomingReset: BOOL := FALSE;

    //Two resets required due to homing functionality
    bResetInProgressCheck1: BOOL := FALSE;
    bResetInProgressCheck2: BOOL := FALSE;

    //internal MCPOWER blocks because Beckhoff won't let you enable a setpoint generator on a limit....
    fbPowerPositiveAxis: MC_POWER;
    fbPowerNegativeAxis: MC_POWER;
    fbPowerGapSizeAxis: MC_POWER;
    fbPowerGapCentreAxis: MC_POWER;

    //internal MC_Reset, needed because the current reset in FB_Axis works only when there is an error. This should change once the reset functionality changes
    fbInternalResetTrig: R_TRIG;
    fbInternalResetHome: R_TRIG;
    fbResetPositiveAxis: MC_RESET;
    fbResetNegativeAxis: MC_RESET;
    fbResetGapSizeAxis: MC_RESET;
    fbResetGapCentreAxis: MC_RESET;
    fbResetHomedGap: MC_Home;
    fbResetHomedCentre: MC_Home;

END_VAR


(*SETUP INSTRUCTIONS
Virtual axes:
Encoder type set to Universal
Encoder mask set to 0xFFFFFFFF
Encoder scaling set to match FB
Link nDataIn1 of encoder to FB encoders
Position lag monitoring can be left on*
Dynamics of virtual axes must be configured considering coupled mechanicals (e.g. don't set velocities your real axes can't achieve)
*)

//Position of virtual axes
actVirtualAxisPositions();
//Limit logic
actVirtualAxisLimits();
//Enable Logic - Virtual axes automatically enable when real axes are enabled
actVirtualAxisEnable();
//Call spGenerator FBs
actGeneratorEnableDisable();
//Calculate position setpoints
actCalculateSetpointPositions();
//Calculate velocity setpoints
actCalculateSetpointVelocities();
//Calculate directions
actCalculateSetpointDirections();

//Error state handling - only handle errors that disable motion
IF bEnable AND (GVL.astAxes[nIdPositiveAxis].Axis.Status.ErrorStop OR GVL.astAxes[nIdNegativeAxis].Axis.Status.ErrorStop OR GVL.astAxes[nIdGapSizeAxis].Axis.Status.ErrorStop OR GVL.astAxes[nIdGapCentreAxis].Axis.Status.ErrorStop) THEN
    eState := E_SlitPairStatesV2.eError;
END_IF

//Propagate real axis error to virtual
IF GVL.astAxes[nIdPositiveAxis].Axis.Status.ErrorStop AND (NOT GVL.astAxes[nIdGapSizeAxis].Axis.Status.ErrorStop OR NOT GVL.astAxes[nIdGapCentreAxis].Axis.Status.ErrorStop) THEN
    GVL.astAxes[nIdGapSizeAxis].stStatus.bError := TRUE;
    GVL.astAxes[nIdGapCentreAxis].stStatus.bError := TRUE;
    GVL.astAxes[nIdGapSizeAxis].stStatus.nErrorID := GVL.astAxes[nIdPositiveAxis].stStatus.nErrorID;
    GVL.astAxes[nIdGapCentreAxis].stStatus.nErrorID := GVL.astAxes[nIdPositiveAxis].stStatus.nErrorID;
ELSIF  GVL.astAxes[nIdNegativeAxis].Axis.Status.ErrorStop AND (NOT GVL.astAxes[nIdGapSizeAxis].Axis.Status.ErrorStop OR NOT GVL.astAxes[nIdGapCentreAxis].Axis.Status.ErrorStop) THEN
    GVL.astAxes[nIdGapSizeAxis].stStatus.bError := TRUE;
    GVL.astAxes[nIdGapCentreAxis].stStatus.bError := TRUE;
    GVL.astAxes[nIdGapSizeAxis].stStatus.nErrorID := GVL.astAxes[nIdNegativeAxis].stStatus.nErrorID;
    GVL.astAxes[nIdGapCentreAxis].stStatus.nErrorID := GVL.astAxes[nIdNegativeAxis].stStatus.nErrorID;
END_IF

//Internal Reset linked to any axis reset
bInternalReset := bReset OR GVL.astAxes[nIdPositiveAxis].stControl.bReset OR GVL.astAxes[nIdNegativeAxis].stControl.bReset OR GVL.astAxes[nIdGapSizeAxis].stControl.bReset OR GVL.astAxes[nIdGapCentreAxis].stControl.bReset;

//If real axis is homing, change state
IF bEnable AND (GVL.astAxes[nIdPositiveAxis].Axis.Status.HomingBusy OR GVL.astAxes[nIdNegativeAxis].Axis.Status.HomingBusy) THEN
    eState := E_SlitPairStatesV2.eWaitForRealHomed;
END_IF

//Link all halt buttons in motors
IF GVL.astAxes[nIdPositiveAxis].stControl.bHalt OR GVL.astAxes[nIdNegativeAxis].stControl.bHalt OR
    GVL.astAxes[nIdGapSizeAxis].stControl.bHalt OR GVL.astAxes[nIdGapCentreAxis].stControl.bHalt THEN
    actHaltAllAxes();
END_IF

//Propagate homing status
fbResetHomedGap(Axis:= GVL.astAxes[nIdGapSizeAxis].Axis, HomingMode:= MC_ResetCalibration);
fbResetHomedCentre(Axis:= GVL.astAxes[nIdGapCentreAxis].Axis, HomingMode:= MC_ResetCalibration);
fbInternalResetHome(CLK:= fbResetHomedCentre.Done OR fbResetHomedGap.Done );
IF NOT GVL.astAxes[nIdPositiveAxis].stStatus.bHomed OR NOT GVL.astAxes[nIdNegativeAxis].stStatus.bHomed THEN
        fbResetHomedGap.Execute := TRUE;
        fbResetHomedCentre.Execute := TRUE;
END_IF

IF fbInternalResetHome.Q THEN
        fbResetHomedGap.Execute := FALSE;
        fbResetHomedCentre.Execute := FALSE;
END_IF


//State machine
IF bEnable THEN
    CASE eState OF  //HOMING LOOP ISSUE
        E_SlitPairStatesV2.eInit:
            //If real axes are calibrated, then home the virtual axes, else go Operatioanl
            fbResetPositiveAxis(Axis:=GVL.astAxes[nIdPositiveAxis].Axis, Execute:=FALSE);
            fbResetNegativeAxis(Axis:=GVL.astAxes[nIdNegativeAxis].Axis, Execute:=FALSE);
            fbResetGapSizeAxis(Axis:=GVL.astAxes[nIdGapSizeAxis].Axis, Execute:=FALSE);
            fbResetGapCentreAxis(Axis:=GVL.astAxes[nIdGapCentreAxis].Axis, Execute:=FALSE);
            IF GVL.astAxes[nIdPositiveAxis].stStatus.bHomed AND GVL.astAxes[nIdNegativeAxis].stStatus.bHomed THEN
               GVL.astAxes[nIdGapSizeAxis].stConfig.eHomeSeq := E_HomingRoutines.eHomeDirect;
               GVL.astAxes[nIdGapCentreAxis].stConfig.eHomeSeq := E_HomingRoutines.eHomeDirect;
               GVL.astAxes[nIdGapSizeAxis].stConfig.fHomePosition := fGapSize;
               GVL.astAxes[nIdGapCentreAxis].stConfig.fHomePosition := fGapCentre;
                eState := E_SlitPairStatesV2.eWaitForVirtualHomed;
            ELSE
                eState := E_SlitPairStatesV2.eOperational;
            END_IF

        E_SlitPairStatesV2.eWaitForVirtualHomed:
            //Wait for virtual axis homing to complete/
            GVL.astAxes[nIdGapSizeAxis].stControl.eCommand := E_MotionFunctions.eHome;
            GVL.astAxes[nIdGapSizeAxis].stControl.bExecute := TRUE;
            GVL.astAxes[nIdGapCentreAxis].stControl.eCommand := E_MotionFunctions.eHome;
            GVL.astAxes[nIdGapCentreAxis].stControl.bExecute := TRUE;
            IF GVL.astAxes[nIdGapSizeAxis].stStatus.bHomed AND GVL.astAxes[nIdGapCentreAxis].stStatus.bHomed THEN
                eState := E_SlitPairStatesV2.eOperational;
            END_IF
            //IF NOT IN HOMING STATE

        E_SlitPairStatesV2.eOperational:
            bResetInProgressCheck1 := FALSE;
            //Detect whether real or virtual axes are moving
            IF GVL.astAxes[nIdGapSizeAxis].stStatus.bMoving OR GVL.astAxes[nIdGapCentreAxis].stStatus.bMoving THEN
                eState := E_SlitPairStatesV2.eEnableRealGenerators;
            END_IF
            IF GVL.astAxes[nIdPositiveAxis].stStatus.bMoving OR GVL.astAxes[nIdNegativeAxis].stStatus.bMoving THEN
                eState := E_SlitPairStatesV2.eEnableVirtualGenerators;
            END_IF

        E_SlitPairStatesV2.eEnableRealGenerators:
            //Hold MC_Power on until generators have enabled
            fbPowerPositiveAxis(Axis:=GVL.astAxes[nIdPositiveAxis].Axis, Enable:=TRUE, Enable_Positive:=TRUE,Enable_Negative:=TRUE);
            fbPowerNegativeAxis(Axis:=GVL.astAxes[nIdNegativeAxis].Axis, Enable:=TRUE, Enable_Positive:=TRUE,Enable_Negative:=TRUE);
            fbSetpointGenEnablePositiveAxis.Execute := TRUE;
            fbSetpointGenEnableNegativeAxis.Execute := TRUE;
            eState := E_SlitPairStatesV2.eCheckRealAxisGeneratorsEnabled;

        E_SlitPairStatesV2.eCheckRealAxisGeneratorsEnabled:
            //Hold MC_Power on until generators have enabled
            fbPowerPositiveAxis(Axis:=GVL.astAxes[nIdPositiveAxis].Axis, Enable:=TRUE, Enable_Positive:=TRUE,Enable_Negative:=TRUE);
            fbPowerNegativeAxis(Axis:=GVL.astAxes[nIdNegativeAxis].Axis, Enable:=TRUE, Enable_Positive:=TRUE,Enable_Negative:=TRUE);
            IF fbSetpointGenEnablePositiveAxis.Enabled AND fbSetpointGenEnableNegativeAxis.Enabled THEN
                eState := E_SlitPairStatesV2.eWaitForVirtualMoveDone;
            END_IF

        E_SlitPairStatesV2.eWaitForVirtualMoveDone:
            IF NOT(GVL.astAxes[nIdGapSizeAxis].stStatus.bMoving OR GVL.astAxes[nIdGapCentreAxis].stStatus.bMoving) THEN
                eState := E_SlitPairStatesV2.eDisableRealGenerators;
            END_IF

        E_SlitPairStatesV2.eDisableRealGenerators:
            fbSetpointGenDisablePositiveAxis.Execute := TRUE;
            fbSetpointGenDisableNegativeAxis.Execute := TRUE;
            eState := E_SlitPairStatesV2.eOperational;

        E_SlitPairStatesV2.eEnableVirtualGenerators:
            //Hold MC_Power on until generators have enabled
            fbPowerGapSizeAxis(Axis:=GVL.astAxes[nIdGapSizeAxis].Axis, Enable:=TRUE, Enable_Positive:=TRUE,Enable_Negative:=TRUE);
            fbPowerGapCentreAxis(Axis:=GVL.astAxes[nIdGapCentreAxis].Axis, Enable:=TRUE, Enable_Positive:=TRUE,Enable_Negative:=TRUE);
            fbSetpointGenEnableGapSizeAxis.Execute := TRUE;
            fbSetpointGenEnableGapCentreAxis.Execute := TRUE;
            eState := E_SlitPairStatesV2.eCheckVirtualAxisGeneratorsEnabled;

        E_SlitPairStatesV2.eCheckVirtualAxisGeneratorsEnabled:
            //Hold MC_Power on until generators have enabled
            fbPowerGapSizeAxis(Axis:=GVL.astAxes[nIdGapSizeAxis].Axis, Enable:=TRUE, Enable_Positive:=TRUE,Enable_Negative:=TRUE);
            fbPowerGapCentreAxis(Axis:=GVL.astAxes[nIdGapCentreAxis].Axis, Enable:=TRUE, Enable_Positive:=TRUE,Enable_Negative:=TRUE);
            IF fbSetpointGenEnableGapSizeAxis.Enabled AND fbSetpointGenEnableGapCentreAxis.Enabled THEN
                eState := E_SlitPairStatesV2.eWaitForRealMoveDone;
            END_IF

        E_SlitPairStatesV2.eWaitForRealMoveDone:
            IF NOT(GVL.astAxes[nIdPositiveAxis].stStatus.bMoving OR GVL.astAxes[nIdNegativeAxis].stStatus.bMoving) THEN
                eState := E_SlitPairStatesV2.eDisableVirtualGenerators;
            END_IF

        E_SlitPairStatesV2.eDisableVirtualGenerators:
            fbSetpointGenDisableGapSizeAxis.Execute := TRUE;
            fbSetpointGenDisableGapCentreAxis.Execute := TRUE;
            eState := E_SlitPairStatesV2.eOperational;

        E_SlitPairStatesV2.eError:
            actHaltAllAxes();

            IF bHomingReset THEN
                bInternalReset := TRUE;
                bResetInProgressCheck1 := TRUE;
                bResetInProgressCheck2 := TRUE;
                bHomingReset := FALSE;
            END_IF
            IF bInternalReset OR bReset OR bResetInProgressCheck2 THEN
                fbResetPositiveAxis(Axis:=GVL.astAxes[nIdPositiveAxis].Axis, Execute:=TRUE);
                fbResetNegativeAxis(Axis:=GVL.astAxes[nIdNegativeAxis].Axis, Execute:=TRUE);
                fbResetGapSizeAxis(Axis:=GVL.astAxes[nIdGapSizeAxis].Axis, Execute:=TRUE);
                fbResetGapCentreAxis(Axis:=GVL.astAxes[nIdGapCentreAxis].Axis, Execute:=TRUE);
                GVL.astAxes[nIdPositiveAxis].stControl.bReset := TRUE;
                GVL.astAxes[nIdNegativeAxis].stControl.bReset := TRUE;
                GVL.astAxes[nIdGapSizeAxis].stControl.bReset := TRUE;
                GVL.astAxes[nIdGapCentreAxis].stControl.bReset := TRUE;
                IF NOT(bResetInProgressCheck1) THEN
                    bResetInProgressCheck2 := FALSE;
                END_IF
            END_IF

            IF NOT(GVL.astAxes[nIdPositiveAxis].stStatus.bError) AND NOT(GVL.astAxes[nIdNegativeAxis].stStatus.bError) AND NOT(GVL.astAxes[nIdGapSizeAxis].stStatus.bError) AND NOT(GVL.astAxes[nIdGapCentreAxis].stStatus.bError) THEN
                eState := E_SlitPairStatesV2.eInit;
            END_IF

        E_SlitPairStatesV2.eWaitForRealHomed:
            bHomingReset := TRUE;
            IF NOT GVL.astAxes[nIdPositiveAxis].Axis.Status.Homed OR NOT GVL.astAxes[nIdNegativeAxis].Axis.Status.Homed THEN
                eState := E_SlitPairStatesV2.eInit;
            END_IF
    END_CASE
END_IF


//Feed externalsetpoint generators setpoint values - ignoring acceleration
MC_ExtSetPointGenFeed(Axis:= GVL.astAxes[nIdPositiveAxis].Axis, Position:= fPosSetpointPositiveAxis, Velocity:= fVeloSetpointPositiveAxis, Acceleration:= 0, Direction:= nDirectionPositiveAxis);
MC_ExtSetPointGenFeed(Axis:= GVL.astAxes[nIdNegativeAxis].Axis, Position:= fPosSetpointNegativeAxis, Velocity:= fVeloSetpointNegativeAxis, Acceleration:= 0, Direction:= nDirectionNegativeAxis);
MC_ExtSetPointGenFeed(Axis:= GVL.astAxes[nIdGapSizeAxis].Axis, Position:= fPosSetpointGapSizeAxis, Velocity:= fVeloSetpointGapSizeAxis, Acceleration:= 0, Direction:= nDirectionGapSizeAxis);
MC_ExtSetPointGenFeed(Axis:= GVL.astAxes[nIdGapCentreAxis].Axis, Position:= fPosSetpointGapCentreAxis, Velocity:= fVeloSetpointGapCentreAxis, Acceleration:= 0, Direction:= nDirectionGapCentreAxis);

bReset := FALSE;

ACTION actCalculateSetpointDirections:

IF fVeloSetpointPositiveAxis > 0 THEN
    nDirectionPositiveAxis := 1; //moving forward
ELSIF fVeloSetpointPositiveAxis < 0 THEN
    nDirectionPositiveAxis := -1; //moving backward
ELSE
    nDirectionPositiveAxis := 0; //stationary
END_IF

IF fVeloSetpointNegativeAxis > 0 THEN
    nDirectionNegativeAxis := 1; //moving forward
ELSIF fVeloSetpointNegativeAxis < 0 THEN
    nDirectionNegativeAxis := -1; //moving backward
ELSE
    nDirectionNegativeAxis := 0; //stationary
END_IF

IF fVeloSetpointGapSizeAxis > 0 THEN
    nDirectionGapSizeAxis := 1; //moving forward
ELSIF fVeloSetpointGapSizeAxis < 0 THEN
    nDirectionGapSizeAxis := -1; //moving backward
ELSE
    nDirectionGapSizeAxis := 0; //stationary
END_IF

IF fVeloSetpointGapCentreAxis > 0 THEN
    nDirectionGapCentreAxis := 1; //moving forward
ELSIF fVeloSetpointGapCentreAxis < 0 THEN
    nDirectionGapCentreAxis := -1; //moving backward
ELSE
    nDirectionGapCentreAxis := 0; //stationary
END_IF
END_ACTION

ACTION actCalculateSetpointPositions:

fPosSetpointPositiveAxis := GVL.astAxes[nIdGapCentreAxis].Axis.NcToPlc.SetPos + (GVL.astAxes[nIdGapSizeAxis].Axis.NcToPlc.SetPos/2);
fPosSetpointNegativeAxis := GVL.astAxes[nIdGapCentreAxis].Axis.NcToPlc.SetPos - (GVL.astAxes[nIdGapSizeAxis].Axis.NcToPlc.SetPos/2);
fPosSetpointGapSizeAxis := GVL.astAxes[nIdPositiveAxis].Axis.NcToPlc.SetPos - GVL.astAxes[nIdNegativeAxis].Axis.NcToPlc.SetPos;
fPosSetpointGapCentreAxis := (GVL.astAxes[nIdPositiveAxis].Axis.NcToPlc.SetPos + GVL.astAxes[nIdNegativeAxis].Axis.NcToPlc.SetPos) / 2;
END_ACTION

ACTION actCalculateSetpointVelocities:

fVeloSetpointPositiveAxis := GVL.astAxes[nIdGapCentreAxis].Axis.NcToPlc.SetVelo +(GVL.astAxes[nIdGapSizeAxis].Axis.NcToPlc.SetVelo/2);
fVeloSetpointNegativeAxis := GVL.astAxes[nIdGapCentreAxis].Axis.NcToPlc.SetVelo -(GVL.astAxes[nIdGapSizeAxis].Axis.NcToPlc.SetVelo/2);
fVeloSetpointGapSizeAxis := GVL.astAxes[nIdPositiveAxis].Axis.NcToPlc.SetVelo - GVL.astAxes[nIdNegativeAxis].Axis.NcToPlc.SetVelo;
fVeloSetpointGapCentreAxis := GVL.astAxes[nIdPositiveAxis].Axis.NcToPlc.SetVelo + GVL.astAxes[nIdNegativeAxis].Axis.NcToPlc.SetVelo;
END_ACTION

ACTION actGeneratorEnableDisable:

fbSetpointGenEnablePositiveAxis(Axis:=GVL.astAxes[nIdPositiveAxis].Axis);
fbSetpointGenEnablePositiveAxis.Execute := FALSE;

fbSetpointGenEnableNegativeAxis(Axis:=GVL.astAxes[nIdNegativeAxis].Axis);
fbSetpointGenEnableNegativeAxis.Execute := FALSE;

fbSetpointGenEnableGapSizeAxis(Axis:=GVL.astAxes[nIdGapSizeAxis].Axis);
fbSetpointGenEnableGapSizeAxis.Execute := FALSE;

fbSetpointGenEnableGapCentreAxis(Axis:=GVL.astAxes[nIdGapCentreAxis].Axis);
fbSetpointGenEnableGapCentreAxis.Execute := FALSE;


fbSetpointGenDisablePositiveAxis(Axis:=GVL.astAxes[nIdPositiveAxis].Axis);
fbSetpointGenDisablePositiveAxis.Execute := FALSE;

fbSetpointGenDisableNegativeAxis(Axis:=GVL.astAxes[nIdNegativeAxis].Axis);
fbSetpointGenDisableNegativeAxis.Execute := FALSE;

fbSetpointGenDisableGapSizeAxis(Axis:=GVL.astAxes[nIdGapSizeAxis].Axis);
fbSetpointGenDisableGapSizeAxis.Execute := FALSE;

fbSetpointGenDisableGapCentreAxis(Axis:=GVL.astAxes[nIdGapCentreAxis].Axis);
fbSetpointGenDisableGapCentreAxis.Execute := FALSE;
END_ACTION

ACTION actHaltAllAxes:

GVL.astAxes[nIdPositiveAxis].stControl.bHalt := TRUE;
GVL.astAxes[nIdNegativeAxis].stControl.bHalt := TRUE;
GVL.astAxes[nIdGapSizeAxis].stControl.bHalt := TRUE;
GVL.astAxes[nIdGapCentreAxis].stControl.bHalt := TRUE;
bAllHalted := TRUE;

//Reset Halts
IF bAllHalted AND NOT GVL.astAxes[nIdPositiveAxis].stStatus.bMoving AND NOT GVL.astAxes[nIdNegativeAxis].stStatus.bMoving
 AND NOT GVL.astAxes[nIdGapSizeAxis].stStatus.bMoving AND NOT GVL.astAxes[nIdGapCentreAxis].stStatus.bMoving THEN
   GVL.astAxes[nIdPositiveAxis].stControl.bHalt := FALSE;
   GVL.astAxes[nIdNegativeAxis].stControl.bHalt := FALSE;
   GVL.astAxes[nIdGapSizeAxis].stControl.bHalt := FALSE;
   GVL.astAxes[nIdGapCentreAxis].stControl.bHalt := FALSE;
   bAllHalted := FALSE;
END_IF
END_ACTION

ACTION actVirtualAxisEnable:

GVL.astAxes[nIdGapSizeAxis].stControl.bEnable := GVL.astAxes[nIdPositiveAxis].stStatus.bEnabled AND GVL.astAxes[nIdNegativeAxis].stStatus.bEnabled;
GVL.astAxes[nIdGapCentreAxis].stControl.bEnable := GVL.astAxes[nIdPositiveAxis].stStatus.bEnabled AND GVL.astAxes[nIdNegativeAxis].stStatus.bEnabled;
END_ACTION

ACTION actVirtualAxisLimits:

GVL.astAxes[nIdGapSizeAxis].stInputs.bLimitFwd := GVL.astAxes[nIdPositiveAxis].stStatus.bFwEnabled AND GVL.astAxes[nIdNegativeAxis].stStatus.bBwEnabled;
GVL.astAxes[nIdGapSizeAxis].stInputs.bLimitBwd := GVL.astAxes[nIdPositiveAxis].stStatus.bBwEnabled AND GVL.astAxes[nIdNegativeAxis].stStatus.bFwEnabled;

GVL.astAxes[nIdGapCentreAxis].stInputs.bLimitFwd := GVL.astAxes[nIdPositiveAxis].stStatus.bFwEnabled AND GVL.astAxes[nIdNegativeAxis].stStatus.bFwEnabled;
GVL.astAxes[nIdGapCentreAxis].stInputs.bLimitBwd := GVL.astAxes[nIdPositiveAxis].stStatus.bBwEnabled AND GVL.astAxes[nIdNegativeAxis].stStatus.bBwEnabled;
END_ACTION

ACTION actVirtualAxisPositions:

(*Calculate virtual axis positions and convert to UDINT.
Conversion to UDINT is prohibited if it would exceed UDINT max value of 4,294,967,295.
If this is not done, it can cause overflow when connected to the encoder input and hard-crash the PLC which will only recover with a power cycle.
To preserve decimal position data of the LREAL (i.e. anything <1mm) it is necessary to scale the value before converting to UDINT.
This can be reversed with the correct scaling at the NC encoder level.
*)
fGapSize := GVL.astAxes[nIdPositiveAxis].stStatus.fActPosition - GVL.astAxes[nIdNegativeAxis].stStatus.fActPosition;
fGapCentre := (GVL.astAxes[nIdPositiveAxis].stStatus.fActPosition + GVL.astAxes[nIdNegativeAxis].stStatus.fActPosition)/2;


    IF ABS(fGapSize) < 100000 THEN
        nGapSizeEncoder := LREAL_TO_UDINT(fGapSize*fEncoderScaling);
    END_IF
    IF ABS(fGapCentre) < 100000 THEN
        nGapCentreEncoder := LREAL_TO_UDINT(fGapCentre*fEncoderScaling);
    END_IF
END_ACTION

END_FUNCTION_BLOCK

// ---- GlobalTextList.TcGTLO
TEXTLIST GlobalTextList
  972 = '  bLocalMode'
  951 = '%2.2f'
  543 = '%2.4f'
  982 = '%d'
  821 = '%s'
  940 = '%x'
  952 = 'actPos'
  953 = 'actVel'
  110 = 'AXESMAX'
  107 = 'axisSel'
  945 = 'bBusy'
  950 = 'bBwEnabled'
  225 = 'bCommandAborted'
  946 = 'bDone'
  943 = 'bEnabled'
  941 = 'bError'
  999 = 'bExtended'
  949 = 'bFwEnabled'
  297 = 'bGeared'
  902 = 'bHighTempAxisDisabled'
  948 = 'bHomed'
  509 = 'bHWMaskActive'
  183 = 'bInterlock'
  512 = 'bInVelocity'
  386 = 'bMoving'
  485 = 'bMovingExtend'
  998 = 'bMovingRetract'
  963 = 'bPSSPermit'
  352 = 'bReset'
  226 = 'bRetracted'
  933 = 'bValveOn'
  786 = 'Bwd Enable'
  350 = 'eHomeDirect'
  302 = 'eHomeToBlock_Bwd'
  1049 = 'eHomeToBlock_Fwd'
  198 = 'eHomeToEncPulse_Bwd'
  510 = 'eHomeToEncPulse_Fwd'
  287 = 'eHomeToEncPulse_viaBwdLimit'
  683 = 'eHomeToEncPulse_viaFwdLimit'
  312 = 'eHomeToLimit_Bwd'
  635 = 'eHomeToLimit_Fwd'
  150 = 'eHomeToRef_Bwd'
  861 = 'eHomeToRef_Fwd'
  87 = 'Elapsed time (ms)'
  104 = 'ENABLE'
  1009 = 'End switches simulation'
  554 = 'EndSwitchBwd'
  1084 = 'EndSwitchFwd'
  1004 = 'eReadParameter'
  939 = 'errID'
  768 = 'eWriteParameter'
  937 = 'E_PneumaticErrors'
  333 = 'E_PneumaticMode'
  955 = 'fAcceleration'
  730 = 'fActualTemp'
  956 = 'fDeceleration'
  531 = 'fHomeFinishDistance'
  613 = 'fHomePosition'
  957 = 'fPosition'
  149 = 'fRatio'
  781 = 'fReadAxisParameter'
  954 = 'fVelocity'
  668 = 'Fwd Enable'
  688 = 'fWriteAxisParameter'
  717 = 'gearInMultiMaster'
  300 = 'gearOut'
  523 = 'halt'
  568 = 'Home'
  784 = 'Interlock Bwd'
  505 = 'Interlock Fwd'
  116 = 'jogBw'
  117 = 'jogFw'
  460 = 'Mode Selection'
  111 = 'moveAbsolute'
  114 = 'moveModulo'
  113 = 'moveRelative'
  112 = 'moveVelocity'
  575 = 'nIndex'
  992 = 'nTimeToExtend(s)'
  995 = 'nTimeToRetract(s)'
  330 = 'Pneumatic Axis Selection'
  942 = 'reset'
  227 = 'Single Solenoid Manual'
  761 = 'Single Solenoid PLC'
  855 = 'sStatus'
  211 = 'Start Extend'
  259 = 'Start Retract'
  115 = 'stop'
END_TEXTLIST

// ---- tc_mca_std_lib/VISUs/languageSupport.TcTLO
TEXTLIST languageSupport
  axesAvailable = 'PLC Axes available: %d' | Test: 'Alt language'
  velocity = 'Velocity:'
  actposition = 'Actual Position:'
  enable = 'Enable Axis'
  enFW = 'Fwd Enable'
  enBW = 'Bwd Enable'
  axisSel = 'Axis Selected:'
  actVelocity = 'Actual Velocity:'
  errID = 'Error ID:'
  bEnabled = 'Axis Enabled'
  bCommandAborted = 'Command Aborted'
  bBusy = 'Busy'
  bDone = 'Command Done'
  bResetDone = 'Reset Complete'
  bHomed = 'Calibrated'
  bFwEnabled = 'Fwd movement enabled'
  bBwEnabled = 'Bwd movement enabled'
  bError = 'Error'
  fVelocity = 'Target Velocity:'
  fAcceleration = 'Target Accel.:'
  fDeceleration = 'Target Decel.:'
  fPosition = 'Target Position:'
  moveAbsolute = 'Absolute position move'
  toggle = 'Toggle'
  moveVelocity = 'Constant velocity move'
  bExecute = 'Motion function executed'
  moveRelative = 'Relative position move'
  moveModulo = 'Modulo position move'
  reset = 'Reset axis'
  stop = 'Stop motion'
  jogBw = 'Jog Backward'
  jogFw = 'Jog Forward'
  bGeared = 'In Gear'
  masterGear = 'Master Axis'
  gearRatio = 'Gear Ratio'
  gearIn = 'Gear In'
  gearOut = 'Gear Out'
  eHomeToLimit_Bwd = 'Bwd Limit'
  eHomeToLimit_Fwd = 'Fwd Limit'
  eHomeToRef_Bwd = 'Home Switch Bwd '
  eHomeToRef_Fwd = 'Home Switch Fwd '
  eHomeToEncPulse_Bwd = 'Enc Index Bwd '
  eHomeToEncPulse_Fwd = 'Enc Index Fwd'
  eHomeToEncPulse_viaBwdLimit = 'Enc Index via Bwd Limit'
  eHomeToEncPulse_viaFwdLimit = 'Enc Index via Fwd Limit'
  eHomeToBlock_Bwd = 'Home To Block Bwd'
  eHomeToBlock_Fwd = 'Home To Block Fwd'
  eHomeDirect = 'Home Direct'
  fHomePosition = 'Set Pos after Homing'
  fHomeFinishDistance = 'Relative Move after Homing'
  halt = 'Halt Motion'
  bInterlockBwd = 'Interlock Bwd'
  bInterlockFwd = 'Interlock Fwd'
  Home = 'HOME'
  eWriteParameter = 'Write Parameter'
  eReadParameter = 'Read Parameter'
  fWriteAxisParameter = 'Parameter to write'
  fReadAxisParameter = 'Parameter'
  bLocalMode = 'Local Mode'
  bInVelocity = 'Target velocity reached'
  bHighTempAxisDisabled = 'Disabled by High Temp '
  fActualTemp = 'Actual Temp'
  bHWMaskActive = 'HW Mask Active'
  bMoving = 'Moving'
   = ''
END_TEXTLIST

// ---- tc_mca_std_lib/VISUs/MainVisu.TcVIS
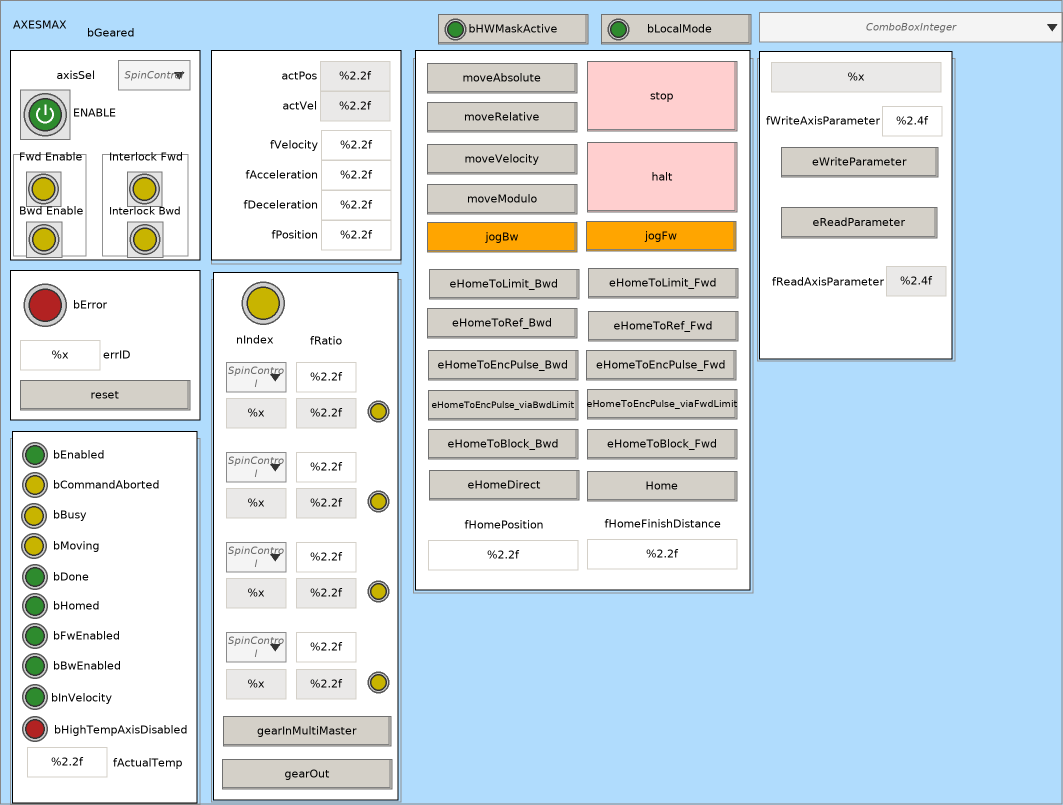
VISUALIZATION MainVisu  // 1063x805
    GroupBox (757,50 198x311)
        Rectangle (2,1 193x308)
        Textfield (14,12 170x30), "%x", text variable: astAxes[MAIN.hmiAxisSelection].stConfig.eAxisParameters
            OnMouseClick: write GVL.astAxes[MAIN.hmiAxisSelection].stConfig.eAxisParameters via Default
        Textfield (6,56 120x30), "fWriteAxisParameter", text list: "languageSupport", text index: "fWriteAxisParameter"
        Textfield (125,56 60x30), "%2.4f", text variable: astAxes[MAIN.hmiAxisSelection].stConfig.fWriteAxisParameter
            OnMouseClick: write GVL.astAxes[MAIN.hmiAxisSelection].stConfig.fWriteAxisParameter via Default
        Button (24,97 157x30), "eWriteParameter", input disabled if: GVL.astAxes[MAIN.hmiAxisSelection].stStatus.bGeared, text list: "languageSupport", text index: "eWriteParameter"
            OnMouseClick: execute { GVL.astAxes[MAIN.hmiAxisSelection].stControl.eCommand:=E_MotionFunctions.eWriteParameter; GVL.astAxes[MAIN.hmiAxisSelection].stControl.bExecute:=TRUE; }
        Button (24,157 156x31), "eReadParameter", input disabled if: GVL.astAxes[MAIN.hmiAxisSelection].stStatus.bGeared, text list: 'languageSupport', text index: "eReadParameter"
            OnMouseClick: execute { GVL.astAxes[MAIN.hmiAxisSelection].stControl.eCommand:=E_MotionFunctions.eReadParameter; GVL.astAxes[MAIN.hmiAxisSelection].stControl.bExecute:=TRUE; }
        Textfield (10,217 120x30), "fReadAxisParameter", text list: "languageSupport", text index: "fReadAxisParameter"
        Textfield (129,216 60x30), "%2.4f", text variable: astAxes[MAIN.hmiAxisSelection].stConfig.fReadAxisParameter
            OnMouseClick: write GVL.astAxes[MAIN.hmiAxisSelection].stConfig.fReadAxisParameter via Default
    GroupBox (413,50 340x543)
        Rectangle (2,0 335x540)
        Button (174,92 150x70), "halt", pressed state: GVL.astAxes[Main.hmiAxisSelection].stControl.bHalt, input disabled if: GVL.astAxes[MAIN.hmiAxisSelection].stStatus.bGeared, text list: "languageSupport", text index: "halt"
            toggle GVL.astAxes[Main.hmiAxisSelection].stControl.bHalt
        Button (174,421 150x30), "Home", input disabled if: GVL.astAxes[MAIN.hmiAxisSelection].stStatus.bGeared, text list: 'languageSupport', text index: "Home"
            OnMouseClick: execute { GVL.astAxes[Main.hmiAxisSelection].stControl.eCommand:=E_MotionFunctions.eHome; GVL.astAxes[Main.hmiAxisSelection].stControl.bExecute:=TRUE; }
        Button (15,379 150x30), "eHomeToBlock_Bwd", input disabled if: GVL.astAxes[MAIN.hmiAxisSelection].stStatus.bGeared, text list: 'languageSupport', text index: "eHomeToBlock_Bwd"
            OnMouseClick: execute {
                GVL.astAxes[Main.hmiAxisSelection].stControl.eCommand:=E_MotionFunctions.eHome;
                GVL.astAxes[Main.hmiAxisSelection].stConfig.eHomeSeq:=E_HomingRoutines.eHomeToBlock_Bwd;
                GVL.astAxes[Main.hmiAxisSelection].stControl.bExecute:=TRUE;
            }
        Button (14,258 150x30), "eHomeToRef_Bwd", input disabled if: GVL.astAxes[MAIN.hmiAxisSelection].stStatus.bGeared, text list: 'languageSupport', text index: "eHomeToRef_Bwd"
            OnMouseClick: execute {
                GVL.astAxes[Main.hmiAxisSelection].stControl.eCommand:=E_MotionFunctions.eHome;
                GVL.astAxes[Main.hmiAxisSelection].stConfig.eHomeSeq:=E_HomingRoutines.eHomeToRef_Bwd;
                GVL.astAxes[Main.hmiAxisSelection].stControl.bExecute:=TRUE;
            }
        Button (14,13 150x30), "moveAbsolute", text list: "languageSupport", text index: "moveAbsolute"
            OnMouseClick: execute { GVL.astAxes[MAIN.hmiAxisSelection].stControl.eCommand:=E_MotionFunctions.eMoveAbsolute; GVL.astAxes[MAIN.hmiAxisSelection].stControl.bExecute:=TRUE; }
        Button (14,94 150x30), "moveVelocity", input disabled if: GVL.astAxes[MAIN.hmiAxisSelection].stStatus.bGeared, text list: "languageSupport", text index: "moveVelocity"
            OnMouseClick: execute { GVL.astAxes[Main.hmiAxisSelection].stControl.eCommand:=E_MotionFunctions.eMoveVelocity; GVL.astAxes[Main.hmiAxisSelection].stControl.bExecute:=TRUE; }
        Button (14,52 150x30), "moveRelative", input disabled if: GVL.astAxes[MAIN.hmiAxisSelection].stStatus.bGeared, text list: "languageSupport", text index: "moveRelative"
            OnMouseClick: execute { GVL.astAxes[Main.hmiAxisSelection].stControl.eCommand:=E_MotionFunctions.eMoveRelative; GVL.astAxes[Main.hmiAxisSelection].stControl.bExecute:=TRUE; }
        Button (14,134 150x30), "moveModulo", input disabled if: GVL.astAxes[MAIN.hmiAxisSelection].stStatus.bGeared, text list: "languageSupport", text index: "moveModulo"
            OnMouseClick: execute { GVL.astAxes[Main.hmiAxisSelection].stControl.eCommand:=E_MotionFunctions.eMoveModulo; GVL.astAxes[Main.hmiAxisSelection].stControl.bExecute:=TRUE; }
        Button (174,11 150x70), "stop", pressed state: GVL.astAxes[Main.hmiAxisSelection].stControl.bStop, input disabled if: GVL.astAxes[MAIN.hmiAxisSelection].stStatus.bGeared, text list: "languageSupport", text index: "stop"
            toggle GVL.astAxes[Main.hmiAxisSelection].stControl.bStop
        Button (14,172 150x30), "jogBw", text list: "languageSupport", text index: "jogBw"
            OnMouseClick: execute {  }
            OnMouseDown: execute {
                GVL.astAxes[Main.hmiAxisSelection].stControl.eCommand:=E_MotionFunctions.eMoveVelocity;
                GVL.astAxes[Main.hmiAxisSelection].stControl.fVelocity:=-ABS(GVL.astAxes[Main.hmiAxisSelection].stControl.fJogVelocity)
                GVL.astAxes[Main.hmiAxisSelection].stControl.bExecute:= TRUE;
            }
            OnMouseUp: execute { GVL.astAxes[Main.hmiAxisSelection].stControl.bHalt:= TRUE; }
        Button (173,171 150x30), "jogFw", text list: "languageSupport", text index: "jogFw"
            OnMouseClick: execute {  }
            OnMouseDown: execute {
                GVL.astAxes[Main.hmiAxisSelection].stControl.eCommand:=E_MotionFunctions.eMoveVelocity;
                GVL.astAxes[Main.hmiAxisSelection].stControl.fVelocity:=ABS(GVL.astAxes[Main.hmiAxisSelection].stControl.fJogVelocity)
                GVL.astAxes[Main.hmiAxisSelection].stControl.bExecute:= TRUE;
            }
            OnMouseUp: execute { GVL.astAxes[Main.hmiAxisSelection].stControl.bHalt:= TRUE; }
        Button (175,261 150x30), "eHomeToRef_Fwd", input disabled if: GVL.astAxes[MAIN.hmiAxisSelection].stStatus.bGeared, text list: "languageSupport", text index: "eHomeToRef_Fwd"
            OnMouseClick: execute {
                GVL.astAxes[Main.hmiAxisSelection].stControl.eCommand:=E_MotionFunctions.eHome;
                GVL.astAxes[Main.hmiAxisSelection].stConfig.eHomeSeq:=E_HomingRoutines.eHomeToRef_Fwd;
                GVL.astAxes[Main.hmiAxisSelection].stControl.bExecute:=TRUE;
            }
        Button (175,218 150x30), "eHomeToLimit_Fwd", input disabled if: GVL.astAxes[MAIN.hmiAxisSelection].stStatus.bGeared, text list: "languageSupport", text index: "eHomeToLimit_Fwd"
            OnMouseClick: execute {
                GVL.astAxes[Main.hmiAxisSelection].stControl.eCommand:=E_MotionFunctions.eHome;
                GVL.astAxes[Main.hmiAxisSelection].stConfig.eHomeSeq:=E_HomingRoutines.eHomeToLimit_Fwd;
                GVL.astAxes[Main.hmiAxisSelection].stControl.bExecute:=TRUE;
            }
        Button (16,219 150x30), "eHomeToLimit_Bwd", input disabled if: GVL.astAxes[MAIN.hmiAxisSelection].stStatus.bGeared, text list: 'languageSupport', text index: "eHomeToLimit_Bwd"
            OnMouseClick: execute {
                GVL.astAxes[Main.hmiAxisSelection].stControl.eCommand:=E_MotionFunctions.eHome;
                GVL.astAxes[Main.hmiAxisSelection].stConfig.eHomeSeq:=E_HomingRoutines.eHomeToLimit_Bwd;
                GVL.astAxes[Main.hmiAxisSelection].stControl.bExecute:=TRUE;
            }
        Button (15,300 150x30), "eHomeToEncPulse_Bwd", input disabled if: GVL.astAxes[MAIN.hmiAxisSelection].stStatus.bGeared, text list: 'languageSupport', text index: "eHomeToEncPulse_Bwd"
            OnMouseClick: execute {
                GVL.astAxes[Main.hmiAxisSelection].stControl.eCommand:=E_MotionFunctions.eHome;
                GVL.astAxes[Main.hmiAxisSelection].stConfig.eHomeSeq:=E_HomingRoutines.eHomeToEncPulse_Bwd;
                GVL.astAxes[Main.hmiAxisSelection].stControl.bExecute:=TRUE;
            }
        Button (173,300 150x30), "eHomeToEncPulse_Fwd", input disabled if: GVL.astAxes[MAIN.hmiAxisSelection].stStatus.bGeared, text list: "languageSupport", text index: "eHomeToEncPulse_Fwd"
            OnMouseClick: execute {
                GVL.astAxes[Main.hmiAxisSelection].stControl.eCommand:=E_MotionFunctions.eHome;
                GVL.astAxes[Main.hmiAxisSelection].stConfig.eHomeSeq:=E_HomingRoutines.eHomeToEncPulse_Fwd;
                GVL.astAxes[Main.hmiAxisSelection].stControl.bExecute:=TRUE;
            }
        Button (174,339 150x30), "eHomeToEncPulse_viaFwdLimit", input disabled if: GVL.astAxes[MAIN.hmiAxisSelection].stStatus.bGeared, text list: "languageSupport", text index: "eHomeToEncPulse_viaFwdLimit"
            OnMouseClick: execute {
                GVL.astAxes[Main.hmiAxisSelection].stControl.eCommand:=E_MotionFunctions.eHome;
                GVL.astAxes[Main.hmiAxisSelection].stConfig.eHomeSeq:=E_HomingRoutines.eHomeToEncPulse_viaFwdLimit;
                GVL.astAxes[Main.hmiAxisSelection].stControl.bExecute:=TRUE;
            }
        Button (15,340 150x30), "eHomeToEncPulse_viaBwdLimit", input disabled if: GVL.astAxes[MAIN.hmiAxisSelection].stStatus.bGeared, text list: 'languageSupport', text index: "eHomeToEncPulse_viaBwdLimit"
            OnMouseClick: execute {
                GVL.astAxes[Main.hmiAxisSelection].stControl.eCommand:=E_MotionFunctions.eHome;
                GVL.astAxes[Main.hmiAxisSelection].stConfig.eHomeSeq:=E_HomingRoutines.eHomeToEncPulse_viaBwdLimit;
                GVL.astAxes[Main.hmiAxisSelection].stControl.bExecute:=TRUE;
            }
        Button (174,379 150x30), "eHomeToBlock_Fwd", input disabled if: GVL.astAxes[MAIN.hmiAxisSelection].stStatus.bGeared, text list: "languageSupport", text index: "eHomeToBlock_Fwd"
            OnMouseClick: execute {
                GVL.astAxes[Main.hmiAxisSelection].stControl.eCommand:=E_MotionFunctions.eHome;
                GVL.astAxes[Main.hmiAxisSelection].stConfig.eHomeSeq:=E_HomingRoutines.eHomeToBlock_Fwd;
                GVL.astAxes[Main.hmiAxisSelection].stControl.bExecute:=TRUE;
            }
        Button (16,420 150x30), "eHomeDirect", input disabled if: GVL.astAxes[MAIN.hmiAxisSelection].stStatus.bGeared, text list: 'languageSupport', text index: "eHomeDirect"
            OnMouseClick: execute {
                GVL.astAxes[Main.hmiAxisSelection].stControl.eCommand:=E_MotionFunctions.eHome;
                GVL.astAxes[Main.hmiAxisSelection].stConfig.eHomeSeq:=E_HomingRoutines.eHomeDirect;
                GVL.astAxes[Main.hmiAxisSelection].stControl.bExecute:=TRUE;
            }
        Textfield (15,490 150x30), "%2.2f", text variable: GVL.astAxes[MAIN.hmiAxisSelection].stConfig.fHomePosition
            OnMouseClick: write the text variable via Default
        Textfield (174,489 150x30), "%2.2f", text variable: GVL.astAxes[MAIN.hmiAxisSelection].stConfig.fHomeFinishDistance, text list: ''
            OnMouseClick: write the text variable via Default
        Textfield (175,459 150x30), "fHomeFinishDistance", text list: "languageSupport", text index: "fHomeFinishDistance"
        Textfield (16,460 150x30), "fHomePosition", text list: "languageSupport", text index: "fHomePosition"
    GroupBox (211,271 190x531)
        Rectangle (2,1 185x528)
        SpinControl (15,91 60x30), variable: GVL.astAxes[MAIN.hmiAxisSelection].stConfig.astMultiMasterAxis[1].nIndex
            p651134158: GVL_APP.nAXIS_NUM
        Textfield (85,91 60x30), "%2.2f", text variable: GVL.astAxes[MAIN.hmiAxisSelection].stConfig.astMultiMasterAxis[1].fRatio
            OnMouseClick: write the text variable via Default
        Textfield (80,55 70x30), "fRatio", text list: "languageSupport", text index: "gearRatio"
        Button (12,445 168x30), "gearInMultiMaster", text list: "languageSupport", text index: "gearIn"
            OnMouseClick: execute { GVL.astAxes[Main.hmiAxisSelection].stControl.eCommand:=E_MotionFunctions.eGearInMultiMaster; GVL.astAxes[Main.hmiAxisSelection].stControl.bExecute:=TRUE; }
        SpinControl (15,181 60x30), variable: GVL.astAxes[MAIN.hmiAxisSelection].stConfig.astMultiMasterAxis[2].nIndex
            p651134158: GVL_APP.nAXIS_NUM
        SpinControl (15,271 60x30), variable: GVL.astAxes[MAIN.hmiAxisSelection].stConfig.astMultiMasterAxis[3].nIndex
            p651134158: GVL_APP.nAXIS_NUM
        SpinControl (15,361 60x30), variable: GVL.astAxes[MAIN.hmiAxisSelection].stConfig.astMultiMasterAxis[4].nIndex
            p651134158: GVL_APP.nAXIS_NUM
        Textfield (85,181 60x30), "%2.2f", text variable: GVL.astAxes[MAIN.hmiAxisSelection].stConfig.astMultiMasterAxis[2].fRatio
            OnMouseClick: write the text variable via Default
        Textfield (85,271 60x30), "%2.2f", text variable: GVL.astAxes[MAIN.hmiAxisSelection].stConfig.astMultiMasterAxis[3].fRatio
            OnMouseClick: write the text variable via Default
        Textfield (85,361 60x30), "%2.2f", text variable: GVL.astAxes[MAIN.hmiAxisSelection].stConfig.astMultiMasterAxis[4].fRatio
            OnMouseClick: write the text variable via Default
        Button (11,488 170x30), "gearOut", text list: "languageSupport", text index: "gearOut"
            OnMouseClick: execute { GVL.astAxes[Main.hmiAxisSelection].stControl.eCommand:=E_MotionFunctions.eGearOut; GVL.astAxes[Main.hmiAxisSelection].stControl.bExecute:=TRUE; }
        Textfield (9,54 70x30), "nIndex", text list: "languageSupport", text index: "masterGear"
        Textfield (85,127 60x30), "%2.2f", text variable: GVL.astAxes[MAIN.hmiAxisSelection].Axis.PlcToNc.GearRatio1
        Textfield (15,127 60x30), "%x", text variable: GVL.astAxes[MAIN.hmiAxisSelection].stConfig.astMultiMasterAxisLatched[1].nIndex
        Textfield (85,217 60x30), "%2.2f", text variable: GVL.astAxes[MAIN.hmiAxisSelection].Axis.PlcToNc.GearRatio2
        Textfield (15,217 60x30), "%x", text variable: GVL.astAxes[MAIN.hmiAxisSelection].stConfig.astMultiMasterAxisLatched[2].nIndex
        Textfield (85,307 60x30), "%2.2f", text variable: GVL.astAxes[MAIN.hmiAxisSelection].Axis.PlcToNc.GearRatio3
        Textfield (15,307 60x30), "%x", text variable: GVL.astAxes[MAIN.hmiAxisSelection].stConfig.astMultiMasterAxisLatched[3].nIndex
        Textfield (85,398 60x30), "%2.2f", text variable: GVL.astAxes[MAIN.hmiAxisSelection].Axis.PlcToNc.GearRatio4
        Textfield (15,398 60x30), "%x", text variable: GVL.astAxes[MAIN.hmiAxisSelection].stConfig.astMultiMasterAxisLatched[4].nIndex
        Lamp1 (155,399 25x25), variable: GVL.astAxes[MAIN.hmiAxisSelection].stStatus.bCoupledGear4, style: Lamp-Lamp1-Yellow
        Lamp1 (155,308 25x25), variable: GVL.astAxes[MAIN.hmiAxisSelection].stStatus.bCoupledGear3, style: Lamp-Lamp1-Yellow
        Lamp1 (155,218 25x25), variable: GVL.astAxes[MAIN.hmiAxisSelection].stStatus.bCoupledGear2, style: Lamp-Lamp1-Yellow
        Lamp1 (155,128 25x25), variable: GVL.astAxes[MAIN.hmiAxisSelection].stStatus.bCoupledGear1, style: Lamp-Lamp1-Yellow
        Lamp1 (27,7 50x50), variable: GVL.astAxes[MAIN.hmiAxisSelection].stStatus.bGeared, style: Lamp-Lamp1-Yellow
    GroupBox (10,50 190x210)
        Rectangle (0,0 190x210)
        GroupBox (3,96 73x110)
        GroupBox (92,96 86x110)
        Textfield (60,50 92x26), "ENABLE", text list: 'languageSupport', text index: "enable"
        PushSwitchLed (16,118 35x42), variable: GVL.astAxes[MAIN.hmiAxisSelection].stInputs.bLimitFwd, behaviour: TOGGLE, style: Switch-PushSwitchLed-Yellow
        PushSwitchLed (16,170 36x39), variable: GVL.astAxes[MAIN.hmiAxisSelection].stInputs.bLimitBwd, behaviour: TOGGLE, style: Switch-PushSwitchLed-Yellow
        SpinControl (108,10 72x30), variable: MAIN.hmiAxisSelection
            p651134158: GVL_APP.nAXIS_NUM
        Textfield (23,13 86x25), "axisSel", text variable: GVL_APP.nAXIS_NUM, text list: "languageSupport", text index: "axisSel"
        PowerSwitch (10,38 50x53), variable: GVL.astAxes[MAIN.hmiAxisSelection].stControl.bEnable, behaviour: TOGGLE, style: Switch-PowerSwitch-Green
        PushSwitchLed (117,118 35x42), variable: GVL.astAxes[MAIN.hmiAxisSelection].stControl.bInterlockFwd, behaviour: TOGGLE, style: Switch-PushSwitchLed-Yellow
        PushSwitchLed (117,170 36x39), variable: GVL.astAxes[MAIN.hmiAxisSelection].stControl.bInterlockBwd, behaviour: TOGGLE, style: Switch-PushSwitchLed-Yellow
        Textfield (6,94 76x26), "Fwd Enable", text list: 'languageSupport', text index: "enFW"
        Textfield (6,148 76x26), "Bwd Enable", text list: 'languageSupport', text index: "enBW"
        Textfield (96,94 76x26), "Interlock Fwd", text list: 'languageSupport', text index: "bAxisInterlockFwd"
        Textfield (96,148 76x26), "Interlock Bwd", text list: 'languageSupport', text index: "bAxisInterlockBwd"
    Textfield (10,10 231x30), "AXESMAX", text variable: GVL_APP.nAXIS_NUM, text list: "languageSupport", text index: "axesAvailable"
    GroupBox (10,270 190x150)
        Rectangle (0,0 190x150)
        Textfield (90,70 90x30), "errID", text list: "languageSupport", text index: "errID"
        Textfield (10,70 80x30), "%x", text variable: GVL.astAxes[MAIN.hmiAxisSelection].stStatus.nErrorID
        Lamp1 (10,10 50x50), variable: GVL.astAxes[MAIN.hmiAxisSelection].stStatus.bError, style: Lamp-Lamp1-Red
        Textfield (60,20 120x30), "bError", text list: "languageSupport", text index: "bError"
        Button (10,110 170x30), "reset", pressed state: GVL.astAxes[Main.hmiAxisSelection].stControl.bReset, text list: "languageSupport", text index: "reset"
            OnMouseClick: toggle GVL.astAxes[Main.hmiAxisSelection].stControl.bReset
    GroupBox (10,430 190x375)
        Rectangle (2,1 185x372)
        Lamp1 (10,10 30x30), variable: GVL.astAxes[MAIN.hmiAxisSelection].stStatus.bEnabled, style: Lamp-Lamp1-Green
        Textfield (40,10 140x30), "bEnabled", text list: "languageSupport", text index: "bEnabled"
        Lamp1 (10,40 30x30), variable: GVL.astAxes[MAIN.hmiAxisSelection].stStatus.bCommandAborted, style: Lamp-Lamp1-Yellow
        Textfield (40,40 140x30), "bCommandAborted", text list: "languageSupport", text index: "bCommandAborted"
        Textfield (40,70 140x30), "bBusy", text list: "languageSupport", text index: "bBusy"
        Lamp1 (10,132 30x30), variable: GVL.astAxes[MAIN.hmiAxisSelection].stStatus.bDone, style: Lamp-Lamp1-Green
        Textfield (40,132 140x30), "bDone", text list: 'languageSupport', text index: "bDone"
        Lamp1 (10,161 30x30), variable: GVL.astAxes[MAIN.hmiAxisSelection].stStatus.bHomed, style: Lamp-Lamp1-Green
        Textfield (40,161 140x30), "bHomed", text list: "languageSupport", text index: "bHomed"
        Lamp1 (10,191 30x30), variable: GVL.astAxes[MAIN.hmiAxisSelection].stStatus.bFwEnabled AND NOT GVL.astAxes[MAIN.hmiAxisSelection].stStatus.bInterlockedFwd, style: Lamp-Lamp1-Green
        Lamp1 (10,221 30x30), variable: GVL.astAxes[MAIN.hmiAxisSelection].stStatus.bBwEnabled AND NOT GVL.astAxes[MAIN.hmiAxisSelection].stStatus.bInterlockedBwd, style: Lamp-Lamp1-Green
        Textfield (40,191 140x30), "bFwEnabled", text list: "languageSupport", text index: "bFwEnabled"
        Textfield (40,221 140x30), "bBwEnabled", text list: "languageSupport", text index: "bBwEnabled"
        Lamp1 (9,71 30x30), variable: GVL.astAxes[MAIN.hmiAxisSelection].stStatus.bBusy, style: Lamp-Lamp1-Yellow
        Lamp1 (10,252 30x30), variable: GVL.astAxes[MAIN.hmiAxisSelection].stStatus.bInVelocity, style: Lamp-Lamp1-Green
        Lamp1 (10,284 30x30), variable: GVL.astAxes[MAIN.hmiAxisSelection].stStatus.bHighTempAxisDisabled, style: Lamp-Lamp1-Red
        Textfield (17,317 80x30), "%2.2f", text variable: GVL.astAxes[MAIN.hmiAxisSelection].stStatus.fActTemperature
        Textfield (100,318 79x30), "fActualTemp", text list: "languageSupport", text index: "fActualTemp"
        Textfield (38,253 140x30), "bInVelocity", text list: 'languageSupport', text index: "bInVelocity"
        Textfield (41,285 140x30), "bHighTempAxisDisabled", text list: 'languageSupport', text index: "bHighTempDisable"
        Lamp1 (9,101 30x30), variable: GVL.astAxes[MAIN.hmiAxisSelection].stStatus.bMoving, style: Lamp-Lamp1-Yellow
        Textfield (40,101 140x30), "bMoving", text list: "languageSupport", text index: "bMoving"
    GroupBox (211,50 190x214)
        Rectangle (0,0 190x210)
        Textfield (10,80 100x30), "fVelocity", text list: "languageSupport", text index: "fVelocity"
        Textfield (110,80 70x30), "%2.2f", text variable: GVL.astAxes[MAIN.hmiAxisSelection].stControl.fVelocity
            OnMouseClick: write the text variable via Default
        Textfield (10,110 100x30), "fAcceleration", text list: "languageSupport", text index: "fAcceleration"
        Textfield (110,110 70x30), "%2.2f", text variable: GVL.astAxes[MAIN.hmiAxisSelection].stControl.fAcceleration
            OnMouseClick: write the text variable via Default
        Textfield (10,140 100x30), "fDeceleration", text list: "languageSupport", text index: "fDeceleration"
        Textfield (110,140 70x30), "%2.2f", text variable: GVL.astAxes[MAIN.hmiAxisSelection].stControl.fDeceleration
            OnMouseClick: write the text variable via Default
        Textfield (10,170 100x30), "fPosition", text list: "languageSupport", text index: "fPosition"
        Textfield (110,170 70x30), "%2.2f", text variable: GVL.astAxes[MAIN.hmiAxisSelection].stControl.fPosition
            OnMouseClick: write the text variable via Default
        Textfield (109,11 70x30), "%2.2f", text variable: GVL.astAxes[MAIN.hmiAxisSelection].stStatus.fActPosition
        Textfield (9,11 100x30), "actPos", text list: "languageSupport", text index: "actposition"
        Textfield (9,41 100x30), "actVel", text list: "languageSupport", text index: "actVelocity"
        Textfield (109,41 70x30), "%2.2f", text variable: GVL.astAxes[MAIN.hmiAxisSelection].stStatus.fActVelocity
        Textfield (-127,-32 93x30), "bGeared", text list: "languageSupport", text index: "bGeared"
    Group (601,14 150x30)
        Button (0,0 150x30), "bLocalMode", text list: 'languageSupport', text index: 'bLocalMode'
            OnMouseClick: toggle bLocalMode
        Lamp1 (5,3 25x25), variable: bLocalMode, style: Lamp-Lamp1-Green
    ComboBoxInteger (759,12 304x30), variable: GVL.astAxes[MAIN.hmiAxisSelection].stConfig.eAxisParameters, text list: 'ParameterTextList'
    Group (438,14 150x30)
        Button (0,0 150x30), "bHWMaskActive", text list: 'languageSupport', text index: 'bHWMaskActive'
            OnMouseClick: toggle bLocalMode
        Lamp1 (5,3 25x25), variable: GVL.astAxes[MAIN.hmiAxisSelection].stControl.bHWMaskActive, style: Lamp-Lamp1-Green
END_VISUALIZATION

// ---- tc_mca_std_lib/VISUs/ParameterTextList.TcTLO
TEXTLIST ParameterTextList
  1 = 'CommandedPosition'
  2 = 'SWLimitForward'
  3 = 'SWLimitBackward'
  4 = 'EnableLimitForward'
  5 = 'EnableLimitBackward'
  6 = 'EnablePositionLagMonitoring'
  7 = 'MaxPositionLag'
  8 = 'AxisMaxVelocity'
  10 = 'ActualVelocity'
  11 = 'CommandedVelocity'
  12 = 'AxisDefaultAcceleration'
  14 = 'AxisDefaultDeceleration'
  16 = 'AxisDefaultJerk'
  1000 = 'AxisId'
  1001 = 'AxisManualVelocitySlow'
  1002 = 'AxisManualVelocityFast'
  1009 = 'AxisRapidTraverseVelocity'
  1012 = 'AxisVelocityToCam'
  1013 = 'AxisVelocityFromCam'
  1014 = 'AxisJogIncrementForward'
  1015 = 'AxisJogIncrementBackward'
  1022 = 'MaxPositionLagFilterTime'
  1023 = 'AxisEnPositionRangeMonitoring'
  1024 = 'AxisPositionRangeWindow'
  1025 = 'AxisEnTargetPositionMonitoring'
  1026 = 'AxisTargetPositionWindow'
  1027 = 'AxisTargetPositionMonitoringTime'
  1028 = 'AxisEnInTargetTimeout'
  1029 = 'AxisInTargetTimeout'
  1030 = 'AxisEnMotionMonitoring'
  1031 = 'AxisMotionMonitoringWindow'
  1032 = 'AxisMotionMonitoringTime'
  1033 = 'AxisDelayTimeVeloPosition'
  1034 = 'AxisEnLoopingDistance'
  1035 = 'AxisLoopingDistance'
  1038 = 'AxisEnDataPersistence'
  1039 = 'AxisRefVeloOnRefOutput'
  1040 = 'AxisOverrideType'
  1042 = 'AxisEncoderOffset'
  1043 = 'AxisEncoderDirectionInverse'
  1044 = 'AxisEncoderMask'
  1045 = 'AxisEncoderModuloValue'
  1046 = 'AxisModuloToleranceWindow'
  1047 = 'AxisEnablePosCorrection'
  1048 = 'AxisPosCorrectionFilterTime'
  1049 = 'AxisUnitInterpretation'
  1050 = 'AxisMotorDirectionInverse'
  1051 = 'AxisCycleTime'
  1052 = 'AxisFastStopSignalType'
  1053 = 'AxisFastAcc'
  1054 = 'AxisFastDec'
  1055 = 'AxisFastJerk'
  1056 = 'AxisEncoderScalingNumerator'
  1057 = 'AxisEncoderScalingDenominator'
  1058 = 'AxisMaximumAcceleration'
  1059 = 'AxisMaximumDeceleration'
  1060 = 'AxisVeloJumpFactor'
  1061 = 'AxisToleranceBallAuxAxis'
  1062 = 'AxisMaxPositionDeviationAuxAxis'
  1063 = 'AxisErrorPropagationMode'
  1064 = 'AxisErrorPropagationDelay'
  1065 = 'AxisCoupleSlaveToActualValues'
  1066 = 'AxisAllowMotionCmdToSlaveAxis'
  1067 = 'AxisAllowMotionCmdToExtSetAxis'
  1068 = 'AxisEncoderSubMask'
  1069 = 'AxisEncoderReferenceSystem'
  1070 = 'AxisEncoderPositionFilterPT1'
  1071 = 'AxisEncoderVelocityFilterPT1'
  1072 = 'AxisEncoderAccelerationFilterPT1'
  1073 = 'AxisEncoderMode'
  1074 = 'AxisEncoderHomingInvDirCamSearch'
  1075 = 'AxisEncoderHomingInvDirSyncSearch'
  1076 = 'AxisEncoderHomingCalibValue'
  1077 = 'AxisEncoderReferenceMode'
  1078 = 'AxisRefVeloOutputRatio'
  1079 = 'AxisDrivePositionOutputScaling'
  1080 = 'AxisDriveVelocityOutputScaling'
  1081 = 'AxisDriveVelocityOutputDelay'
  1082 = 'AxisDriveMinOutputLimitation'
  1083 = 'AxisDriveMaxOutputLimitation'
  1084 = 'AxisTorqueInputScaling'
  1085 = 'AxisTorqueInputFilterPT1'
  1086 = 'AxisTorqueDerivationInputFilterPT1'
  1087 = 'AxisTorqueOutputScaling'
  1088 = 'AxisTorqueOutputDelay'
  1089 = 'AxisAccelerationOutputScaling'
  1090 = 'AxisAccelerationOutputDelay'
  1091 = 'AxisDrivePositionOutputSmoothFilterType'
  1092 = 'AxisDrivePositionOutputSmoothFilterTime'
  1093 = 'AxisDrivePositionOutputSmoothFilterOrder'
  1094 = 'AxisDriveMode'
  1095 = 'AxisDriftCompensationOffset'
  1096 = 'AxisPositionControlKv'
  1097 = 'AxisCtrlVelocityPreCtrlWeight'
  1098 = 'AxisControllerMode'
  1099 = 'AxisCtrlAutoOffset'
  1100 = 'AxisCtrlAutoOffsetTimer'
  1101 = 'AxisCtrlAutoOffsetLimit'
  1102 = 'AxisSlaveCouplingControlKcp'
  1103 = 'AxisCtrlOutputLimit'
  2000 = 'AxisTargetPosition'
  2001 = 'AxisRemainingTimeToGo'
  2002 = 'AxisRemainingDistanceToGo'
  3000 = 'AxisGearRatio'
  4000 = 'NcSafCycleTime'
  4001 = 'NcSvbCycleTime'
   = ''
END_TEXTLIST

